C03641=1051.470,441.160,366.579,176.054,43.114,158.636
C03642=1051.459,440.916,366.630,176.041,43.103,158.631
C03643=1051.447,440.672,366.681,176.027,43.091,158.627
C03644=1051.435,440.427,366.732,176.014,43.081,158.623
C03645=1051.424,440.183,366.784,176.001,43.069,158.619
C03646=1051.413,439.938,366.835,175.987,43.058,158.615
C03647=1051.402,439.694,366.886,175.974,43.047,158.611
C03648=1051.390,439.450,366.937,175.961,43.036,158.607
C03649=1051.379,439.205,366.988,175.949,43.025,158.603
C03650=1051.364,438.882,367.055,175.931,43.011,158.597
C03651=1051.349,438.559,367.122,175.914,42.996,158.592
C03652=1051.334,438.236,367.189,175.897,42.981,158.587
C03653=1051.320,437.914,367.256,175.881,42.967,158.581
C03654=1051.308,437.669,367.307,175.868,42.956,158.577
C03655=1051.297,437.424,367.357,175.854,42.945,158.573
C03656=1051.286,437.180,367.408,175.843,42.935,158.570
C03657=1051.274,436.935,367.459,175.830,42.924,158.566
C03658=1051.263,436.691,367.509,175.818,42.913,158.562
C03659=1051.253,436.446,367.559,175.805,42.902,158.558
C03660=1051.242,436.201,367.609,175.792,42.892,158.554
C03661=1051.230,435.956,367.660,175.780,42.881,158.550
C03662=1051.219,435.712,367.710,175.767,42.871,158.546
C03663=1051.209,435.467,367.760,175.755,42.860,158.542
C03664=1051.198,435.222,367.810,175.742,42.850,158.539
C03665=1051.186,434.978,367.860,175.731,42.839,158.535
C03666=1051.175,434.733,367.910,175.719,42.829,158.531
C03667=1051.164,434.489,367.960,175.706,42.819,158.527
C03668=1051.154,434.244,368.009,175.694,42.808,158.524
C03669=1051.143,433.999,368.060,175.683,42.798,158.520
C03670=1051.132,433.754,368.109,175.670,42.788,158.516
C03671=1051.121,433.509,368.159,175.658,42.778,158.513
C03672=1051.110,433.264,368.208,175.647,42.767,158.509
C03673=1051.099,433.020,368.258,175.635,42.757,158.505
C03674=1051.085,432.691,368.324,175.619,42.743,158.500
C03675=1051.071,432.362,368.391,175.603,42.730,158.495
C03676=1051.057,432.033,368.458,175.588,42.716,158.491
C03677=1051.042,431.704,368.524,175.572,42.702,158.486
C03678=1051.031,431.459,368.573,175.560,42.693,158.482
C03679=1051.020,431.214,368.623,175.549,42.683,158.479
C03680=1051.011,430.969,368.672,175.537,42.672,158.475
C03681=1051.000,430.724,368.721,175.526,42.663,158.472
C03682=1050.989,430.479,368.770,175.514,42.653,158.468
C03683=1050.978,430.235,368.819,175.503,42.643,158.465
C03684=1050.968,429.989,368.868,175.492,42.633,158.461
C03685=1050.958,429.745,368.918,175.480,42.623,158.458
C03686=1050.948,429.499,368.966,175.469,42.613,158.454
C03687=1050.937,429.255,369.015,175.458,42.604,158.451
C03688=1050.927,429.010,369.064,175.447,42.594,158.447
C03689=1050.915,428.764,369.112,175.436,42.584,158.444
C03690=1050.906,428.519,369.161,175.425,42.575,158.440
C03691=1050.894,428.275,369.210,175.414,42.565,158.437
C03692=1050.885,428.030,369.258,175.403,42.555,158.434
C03693=1050.874,427.784,369.307,175.392,42.546,158.430
C03694=1050.864,427.539,369.355,175.380,42.536,158.427
C03695=1050.854,427.294,369.404,175.370,42.526,158.424
C03696=1050.843,427.049,369.452,175.359,42.517,158.420
C03697=1050.833,426.804,369.501,175.348,42.507,158.417
C03698=1050.823,426.559,369.548,175.338,42.498,158.414
C03699=1050.812,426.314,369.597,175.327,42.489,158.411
C03700=1050.802,426.069,369.645,175.316,42.480,158.407
C03701=1050.792,425.823,369.693,175.306,42.470,158.404
C03702=1050.782,425.579,369.741,175.295,42.461,158.401
C03703=1050.772,425.334,369.790,175.285,42.451,158.397
C03704=1050.761,425.088,369.837,175.274,42.442,158.394
C03705=1050.751,424.843,369.886,175.263,42.433,158.391
C03706=1050.741,424.597,369.933,175.253,42.424,158.388
C03707=1050.731,424.353,369.981,175.242,42.415,158.385
C03708=1050.721,424.108,370.028,175.232,42.405,158.382
C03709=1050.710,423.861,370.076,175.221,42.397,158.378
C03710=1050.700,423.617,370.124,175.211,42.387,158.375
C03711=1050.690,423.371,370.171,175.200,42.378,158.372
C03712=1050.680,423.126,370.219,175.191,42.369,158.369
C03713=1050.670,422.880,370.266,175.181,42.360,158.366
C03714=1050.660,422.636,370.314,175.170,42.351,158.363
C03715=1050.649,422.390,370.362,175.160,42.342,158.360
C03716=1050.640,422.145,370.409,175.149,42.333,158.357
C03717=1050.630,421.900,370.457,175.140,42.324,158.354
C03718=1050.620,421.655,370.503,175.130,42.315,158.351
C03719=1050.610,421.410,370.551,175.119,42.307,158.348
C03720=1050.601,421.164,370.598,175.109,42.298,158.345
C03721=1050.590,420.919,370.646,175.100,42.289,158.342
C03722=1050.581,420.673,370.692,175.090,42.280,158.339
C03723=1050.570,420.428,370.739,175.079,42.271,158.335
C03724=1050.561,420.183,370.787,175.070,42.262,158.332
C03725=1050.551,419.937,370.834,175.060,42.253,158.329
C03726=1050.541,419.692,370.881,175.050,42.245,158.327
C03727=1050.531,419.446,370.928,175.041,42.236,158.324
C03728=1050.523,419.201,370.974,175.030,42.228,158.321
C03729=1050.512,418.955,371.022,175.021,42.219,158.318
C03730=1050.496,418.571,371.095,175.006,42.205,158.313
C03731=1050.481,418.186,371.168,174.991,42.192,158.309
C03732=1050.466,417.802,371.240,174.976,42.179,158.304
C03733=1050.451,417.417,371.313,174.961,42.166,158.300
C03734=1050.441,417.171,371.360,174.951,42.157,158.297
C03735=1050.432,416.926,371.406,174.942,42.149,158.294
C03736=1050.422,416.680,371.453,174.933,42.141,158.291
C03737=1050.413,416.434,371.499,174.923,42.132,158.288
C03738=1050.403,416.189,371.546,174.914,42.124,158.286
C03739=1050.393,415.944,371.592,174.904,42.115,158.283
C03740=1050.384,415.697,371.638,174.895,42.107,158.280
C03741=1050.374,415.452,371.684,174.886,42.099,158.277
C03742=1050.365,415.207,371.730,174.877,42.090,158.275
C03743=1050.355,414.961,371.777,174.868,42.082,158.272
C03744=1050.345,414.716,371.822,174.859,42.074,158.269
C03745=1050.335,414.470,371.869,174.849,42.066,158.266
C03746=1050.326,414.225,371.914,174.840,42.057,158.264
C03747=1050.317,413.979,371.960,174.831,42.050,158.261
C03748=1050.308,413.734,372.006,174.821,42.042,158.258
C03749=1050.298,413.488,372.052,174.813,42.033,158.256
C03750=1050.289,413.242,372.098,174.804,42.025,158.253
C03751=1050.280,412.997,372.144,174.795,42.017,158.250
C03752=1050.271,412.751,372.190,174.786,42.009,158.247
C03753=1050.260,412.505,372.235,174.777,42.001,158.245
C03754=1050.251,412.259,372.280,174.768,41.993,158.242
C03755=1050.242,412.014,372.326,174.759,41.986,158.240
C03756=1050.232,411.769,372.371,174.750,41.978,158.237
C03757=1050.223,411.522,372.417,174.742,41.970,158.234
C03758=1050.213,411.277,372.462,174.733,41.962,158.232
C03759=1050.204,411.031,372.508,174.724,41.954,158.229
C03760=1050.195,410.786,372.553,174.715,41.946,158.227
C03761=1050.185,410.540,372.598,174.707,41.939,158.224
C03762=1050.176,410.294,372.644,174.697,41.931,158.222
C03763=1050.166,410.049,372.689,174.689,41.923,158.219
C03764=1050.157,409.803,372.734,174.680,41.915,158.216
C03765=1050.148,409.557,372.779,174.672,41.907,158.214
C03766=1050.139,409.312,372.824,174.663,41.899,158.211
C03767=1050.130,409.065,372.869,174.655,41.892,158.209
C03768=1050.120,408.820,372.914,174.646,41.884,158.206
C03769=1050.111,408.574,372.959,174.638,41.877,158.204
C03770=1050.102,408.328,373.004,174.629,41.869,158.201
C03771=1050.093,408.082,373.049,174.621,41.861,158.199
C03772=1050.083,407.836,373.094,174.612,41.854,158.196
C03773=1050.075,407.591,373.139,174.604,41.846,158.194
C03774=1050.066,407.345,373.184,174.595,41.839,158.191
C03775=1050.056,407.099,373.228,174.588,41.831,158.189
C03776=1050.048,406.853,373.274,174.579,41.824,158.187
C03777=1050.038,406.607,373.318,174.571,41.817,158.184
C03778=1050.030,406.362,373.363,174.562,41.809,158.182
C03779=1050.020,406.116,373.407,174.554,41.801,158.179
C03780=1050.011,405.870,373.452,174.546,41.794,158.177
C03781=1050.003,405.625,373.496,174.537,41.787,158.175
C03782=1049.994,405.378,373.541,174.529,41.779,158.172
C03783=1049.984,405.133,373.585,174.522,41.772,158.170
C03784=1049.976,404.887,373.630,174.513,41.765,158.167
C03785=1049.967,404.641,373.674,174.505,41.757,158.165
C03786=1049.953,404.263,373.742,174.493,41.746,158.161
C03787=1049.939,403.885,373.811,174.480,41.735,158.158
C03788=1049.925,403.507,373.878,174.468,41.724,158.154
C03789=1049.912,403.129,373.946,174.456,41.712,158.151
C03790=1049.903,402.883,373.990,174.447,41.705,158.148
C03791=1049.894,402.637,374.034,174.440,41.698,158.146
C03792=1049.886,402.391,374.079,174.432,41.691,158.144
C03793=1049.876,402.145,374.123,174.424,41.684,158.141
C03794=1049.868,401.899,374.166,174.417,41.677,158.139
C03795=1049.858,401.653,374.210,174.408,41.670,158.137
C03796=1049.850,401.407,374.254,174.400,41.663,158.135
C03797=1049.841,401.161,374.298,174.393,41.656,158.132
C03798=1049.832,400.915,374.341,174.385,41.649,158.130
C03799=1049.823,400.670,374.385,174.377,41.642,158.128
C03800=1049.814,400.423,374.428,174.370,41.635,158.126
C03801=1049.806,400.178,374.472,174.361,41.628,158.123
C03802=1049.796,399.931,374.516,174.354,41.621,158.121
C03803=1049.788,399.685,374.559,174.346,41.614,158.119
C03804=1049.779,399.440,374.603,174.338,41.608,158.117
C03805=1049.770,399.194,374.646,174.331,41.600,158.115
C03806=1049.762,398.947,374.690,174.323,41.594,158.113
C03807=1049.753,398.701,374.734,174.316,41.587,158.110
C03808=1049.745,398.455,374.777,174.308,41.580,158.108
C03809=1049.736,398.209,374.820,174.301,41.573,158.106
C03810=1049.727,397.963,374.864,174.293,41.566,158.104
C03811=1049.718,397.717,374.907,174.286,41.560,158.102
C03812=1049.710,397.471,374.950,174.278,41.553,158.100
C03813=1049.701,397.225,374.993,174.271,41.546,158.097
C03814=1049.692,396.980,375.037,174.263,41.539,158.095
C03815=1049.684,396.734,375.080,174.256,41.533,158.093
C03816=1049.675,396.487,375.123,174.248,41.526,158.091
C03817=1049.667,396.241,375.166,174.241,41.519,158.089
C03818=1049.658,395.995,375.209,174.233,41.513,158.087
C03819=1049.650,395.749,375.252,174.226,41.506,158.085
C03820=1049.641,395.504,375.294,174.219,41.499,158.083
C03821=1049.632,395.258,375.337,174.211,41.493,158.081
C03822=1049.623,395.011,375.381,174.204,41.486,158.078
C03823=1049.615,394.764,375.423,174.196,41.480,158.077
C03824=1049.607,394.519,375.466,174.189,41.473,158.074
C03825=1049.598,394.273,375.508,174.182,41.467,158.072
C03826=1049.589,394.027,375.551,174.175,41.460,158.070
C03827=1049.581,393.781,375.594,174.168,41.454,158.068
C03828=1049.573,393.534,375.637,174.161,41.447,158.066
C03829=1049.564,393.288,375.680,174.153,41.441,158.064
C03830=1049.556,393.042,375.723,174.146,41.435,158.062
C03831=1049.547,392.796,375.764,174.138,41.428,158.060
C03832=1049.538,392.550,375.807,174.131,41.422,158.058
C03833=1049.530,392.304,375.849,174.125,41.415,158.056
C03834=1049.522,392.058,375.892,174.118,41.409,158.054
C03835=1049.513,391.811,375.934,174.110,41.403,158.052
C03836=1049.505,391.565,375.977,174.103,41.396,158.050
C03837=1049.496,391.319,376.019,174.097,41.390,158.048
C03838=1049.487,391.073,376.062,174.090,41.384,158.046
C03839=1049.480,390.827,376.104,174.082,41.377,158.044
C03840=1049.471,390.580,376.146,174.075,41.371,158.042
C03841=1049.462,390.334,376.188,174.068,41.365,158.040
C03842=1049.450,389.975,376.250,174.058,41.356,158.038
C03843=1049.438,389.616,376.311,174.048,41.347,158.035
C03844=1049.426,389.256,376.372,174.038,41.338,158.032
C03845=1049.414,388.897,376.434,174.028,41.329,158.029
C03846=1049.406,388.650,376.476,174.021,41.323,158.027
C03847=1049.397,388.404,376.518,174.014,41.316,158.025
C03848=1049.389,388.157,376.560,174.007,41.310,158.023
C03849=1049.380,387.911,376.601,174.000,41.304,158.022
C03850=1049.371,387.665,376.643,173.994,41.299,158.020
C03851=1049.364,387.419,376.685,173.987,41.292,158.018
C03852=1049.355,387.172,376.726,173.980,41.286,158.016
C03853=1049.346,386.926,376.768,173.974,41.281,158.014
C03854=1049.339,386.680,376.810,173.967,41.274,158.012
C03855=1049.330,386.433,376.851,173.960,41.269,158.011
C03856=1049.322,386.187,376.893,173.953,41.263,158.009
C03857=1049.313,385.940,376.934,173.946,41.256,158.007
C03858=1049.305,385.695,376.976,173.940,41.251,158.005
C03859=1049.297,385.448,377.018,173.933,41.244,158.003
C03860=1049.289,385.202,377.058,173.927,41.239,158.001
C03861=1049.280,384.955,377.100,173.920,41.233,158.000
C03862=1049.273,384.709,377.141,173.913,41.227,157.998
C03863=1049.264,384.462,377.183,173.907,41.221,157.996
C03864=1049.256,384.216,377.224,173.900,41.216,157.994
C03865=1049.248,383.970,377.266,173.894,41.209,157.992
C03866=1049.239,383.723,377.307,173.887,41.204,157.991
C03867=1049.231,383.478,377.348,173.881,41.198,157.989
C03868=1049.224,383.231,377.389,173.874,41.192,157.987
C03869=1049.215,382.985,377.431,173.868,41.186,157.985
C03870=1049.207,382.738,377.472,173.861,41.181,157.983
C03871=1049.200,382.492,377.513,173.855,41.175,157.982
C03872=1049.191,382.245,377.554,173.848,41.169,157.980
C03873=1049.183,381.999,377.595,173.842,41.163,157.978
C03874=1049.175,381.752,377.636,173.836,41.158,157.976
C03875=1049.167,381.505,377.677,173.829,41.152,157.975
C03876=1049.159,381.259,377.718,173.823,41.146,157.973
C03877=1049.150,381.014,377.759,173.816,41.141,157.971
C03878=1049.143,380.767,377.801,173.810,41.135,157.969
C03879=1049.135,380.521,377.841,173.803,41.129,157.968
C03880=1049.126,380.274,377.882,173.797,41.124,157.966
C03881=1049.119,380.027,377.924,173.791,41.118,157.964
C03882=1049.111,379.781,377.964,173.784,41.112,157.963
C03883=1049.103,379.535,378.005,173.778,41.106,157.961
C03884=1049.095,379.288,378.045,173.772,41.101,157.959
C03885=1049.087,379.042,378.086,173.765,41.096,157.957
C03886=1049.079,378.794,378.126,173.760,41.090,157.956
C03887=1049.071,378.548,378.167,173.753,41.085,157.954
C03888=1049.063,378.302,378.208,173.747,41.079,157.952
C03889=1049.055,378.055,378.248,173.741,41.074,157.951
C03890=1049.047,377.809,378.288,173.734,41.068,157.949
C03891=1049.039,377.562,378.329,173.728,41.063,157.948
C03892=1049.031,377.316,378.369,173.722,41.057,157.946
C03893=1049.022,377.068,378.410,173.715,41.052,157.944
C03894=1049.014,376.822,378.450,173.710,41.046,157.942
C03895=1049.006,376.576,378.491,173.704,41.041,157.941
C03896=1048.999,376.329,378.531,173.698,41.036,157.939
C03897=1048.991,376.083,378.572,173.691,41.030,157.938
C03898=1048.980,375.756,378.624,173.684,41.023,157.936
C03899=1048.970,375.430,378.678,173.675,41.016,157.933
C03900=1048.959,375.103,378.731,173.667,41.009,157.931
C03901=1048.949,374.776,378.784,173.660,41.002,157.929
C03902=1048.941,374.530,378.825,173.654,40.997,157.928
C03903=1048.933,374.283,378.865,173.647,40.992,157.926
C03904=1048.925,374.036,378.905,173.641,40.986,157.924
C03905=1048.917,373.790,378.945,173.635,40.981,157.923
C03906=1048.910,373.543,378.985,173.630,40.975,157.921
C03907=1048.902,373.297,379.025,173.624,40.970,157.920
C03908=1048.894,373.050,379.064,173.617,40.965,157.918
C03909=1048.886,372.804,379.105,173.611,40.960,157.916
C03910=1048.878,372.557,379.145,173.606,40.955,157.915
C03911=1048.871,372.310,379.184,173.600,40.949,157.913
C03912=1048.863,372.064,379.224,173.594,40.944,157.912
C03913=1048.856,371.817,379.264,173.588,40.939,157.910
C03914=1048.848,371.570,379.304,173.582,40.934,157.909
C03915=1048.840,371.323,379.344,173.576,40.928,157.907
C03916=1048.832,371.076,379.383,173.570,40.923,157.905
C03917=1048.825,370.830,379.423,173.565,40.918,157.904
C03918=1048.817,370.583,379.463,173.559,40.913,157.902
C03919=1048.809,370.337,379.502,173.553,40.908,157.901
C03920=1048.801,370.090,379.542,173.548,40.903,157.900
C03921=1048.792,369.843,379.581,173.542,40.898,157.898
C03922=1048.786,369.596,379.620,173.535,40.893,157.896
C03923=1048.778,369.349,379.660,173.530,40.888,157.895
C03924=1048.769,369.103,379.699,173.524,40.883,157.893
C03925=1048.762,368.857,379.739,173.518,40.878,157.892
C03926=1048.754,368.609,379.777,173.513,40.873,157.890
C03927=1048.746,368.362,379.817,173.507,40.868,157.889
C03928=1048.738,368.116,379.857,173.501,40.863,157.887
C03929=1048.731,367.869,379.895,173.496,40.858,157.886
C03930=1048.723,367.622,379.935,173.490,40.853,157.885
C03931=1048.716,367.376,379.974,173.485,40.848,157.883
C03932=1048.708,367.129,380.013,173.479,40.843,157.882
C03933=1048.700,366.882,380.053,173.473,40.838,157.880
C03934=1048.693,366.635,380.092,173.468,40.834,157.879
C03935=1048.684,366.389,380.131,173.462,40.828,157.877
C03936=1048.678,366.142,380.170,173.456,40.824,157.876
C03937=1048.669,365.895,380.209,173.451,40.818,157.874
C03938=1048.662,365.648,380.248,173.445,40.814,157.873
C03939=1048.655,365.401,380.287,173.440,40.809,157.871
C03940=1048.646,365.154,380.327,173.434,40.804,157.870
C03941=1048.640,364.908,380.365,173.428,40.799,157.869
C03942=1048.631,364.661,380.405,173.423,40.794,157.867
C03943=1048.624,364.414,380.444,173.417,40.790,157.866
C03944=1048.617,364.168,380.482,173.412,40.785,157.864
C03945=1048.609,363.920,380.521,173.406,40.780,157.863
C03946=1048.602,363.674,380.560,173.401,40.775,157.862
C03947=1048.594,363.427,380.599,173.395,40.770,157.860
C03948=1048.587,363.180,380.637,173.390,40.765,157.859
C03949=1048.579,362.933,380.677,173.385,40.761,157.857
C03950=1048.572,362.686,380.715,173.379,40.756,157.856
C03951=1048.564,362.440,380.753,173.374,40.751,157.854
C03952=1048.557,362.192,380.792,173.368,40.746,157.853
C03953=1048.549,361.946,380.830,173.363,40.742,157.852
C03954=1048.540,361.638,380.879,173.356,40.736,157.850
C03955=1048.529,361.330,380.927,173.349,40.730,157.848
C03956=1048.520,361.023,380.975,173.342,40.724,157.846
C03957=1048.511,360.715,381.023,173.336,40.719,157.845
C03958=1048.504,360.468,381.061,173.331,40.714,157.844
C03959=1048.496,360.222,381.099,173.326,40.710,157.842
C03960=1048.488,359.975,381.138,173.320,40.705,157.841
C03961=1048.480,359.728,381.176,173.315,40.700,157.839
C03962=1048.474,359.481,381.214,173.309,40.696,157.838
C03963=1048.466,359.234,381.253,173.304,40.691,157.837
C03964=1048.458,358.987,381.291,173.299,40.686,157.835
C03965=1048.451,358.741,381.329,173.294,40.682,157.834
C03966=1048.443,358.493,381.367,173.288,40.678,157.833
C03967=1048.436,358.246,381.406,173.283,40.673,157.831
C03968=1048.429,357.999,381.444,173.277,40.669,157.830
C03969=1048.421,357.752,381.482,173.273,40.664,157.829
C03970=1048.414,357.506,381.520,173.268,40.660,157.827
C03971=1048.406,357.258,381.559,173.262,40.655,157.826
C03972=1048.398,357.011,381.596,173.257,40.651,157.825
C03973=1048.391,356.764,381.634,173.252,40.646,157.823
C03974=1048.384,356.518,381.672,173.247,40.642,157.822
C03975=1048.376,356.270,381.710,173.241,40.637,157.821
C03976=1048.368,356.023,381.748,173.236,40.633,157.820
C03977=1048.361,355.776,381.786,173.231,40.628,157.818
C03978=1048.353,355.530,381.824,173.226,40.624,157.817
C03979=1048.346,355.283,381.861,173.221,40.619,157.816
C03980=1048.339,355.035,381.899,173.215,40.615,157.814
C03981=1048.331,354.789,381.937,173.210,40.611,157.813
C03982=1048.323,354.541,381.975,173.206,40.606,157.812
C03983=1048.316,354.294,382.013,173.200,40.602,157.811
C03984=1048.309,354.047,382.050,173.195,40.597,157.809
C03985=1048.301,353.800,382.088,173.191,40.593,157.808
C03986=1048.294,353.553,382.126,173.185,40.589,157.807
C03987=1048.287,353.306,382.163,173.180,40.585,157.806
C03988=1048.280,353.059,382.201,173.175,40.580,157.804
C03989=1048.272,352.812,382.238,173.170,40.575,157.803
C03990=1048.265,352.565,382.277,173.165,40.571,157.802
C03991=1048.258,352.318,382.314,173.161,40.567,157.801
C03992=1048.250,352.071,382.352,173.155,40.563,157.799
C03993=1048.243,351.824,382.389,173.150,40.559,157.798
C03994=1048.236,351.577,382.427,173.146,40.554,157.797
C03995=1048.229,351.330,382.464,173.140,40.550,157.796
C03996=1048.221,351.082,382.502,173.135,40.545,157.794
C03997=1048.214,350.835,382.539,173.130,40.541,157.793
C03998=1048.207,350.588,382.577,173.125,40.537,157.792
C03999=1048.199,350.341,382.614,173.120,40.533,157.791
C04000=1048.192,350.094,382.651,173.115,40.528,157.789
C04001=1048.185,349.846,382.688,173.110,40.524,157.788
C04002=1048.178,349.599,382.726,173.106,40.520,157.787
C04003=1048.170,349.352,382.763,173.101,40.516,157.786
C04004=1048.163,349.106,382.800,173.095,40.512,157.785
C04005=1048.156,348.858,382.837,173.091,40.508,157.783
C04006=1048.149,348.611,382.874,173.086,40.503,157.782
C04007=1048.141,348.364,382.911,173.081,40.499,157.781
C04008=1048.134,348.117,382.949,173.076,40.495,157.780
C04009=1048.127,347.869,382.985,173.071,40.491,157.779
C04010=1048.117,347.568,383.031,173.065,40.486,157.777
C04011=1048.108,347.265,383.076,173.060,40.481,157.776
C04012=1048.100,346.963,383.121,173.053,40.476,157.774
C04013=1048.092,346.661,383.166,173.048,40.471,157.773
C04014=1048.084,346.415,383.203,173.043,40.467,157.772
C04015=1048.076,346.167,383.241,173.038,40.462,157.770
C04016=1048.069,345.920,383.277,173.033,40.459,157.769
C04017=1048.062,345.672,383.314,173.029,40.454,157.768
C04018=1048.055,345.426,383.351,173.023,40.450,157.767
C04019=1048.047,345.178,383.387,173.019,40.446,157.766
C04020=1048.040,344.931,383.424,173.014,40.442,157.765
C04021=1048.033,344.683,383.461,173.010,40.438,157.764
C04022=1048.026,344.437,383.498,173.005,40.434,157.762
C04023=1048.019,344.190,383.535,173.000,40.430,157.761
C04024=1048.011,343.942,383.571,172.995,40.426,157.760
C04025=1048.005,343.696,383.608,172.991,40.422,157.759
C04026=1047.997,343.448,383.644,172.986,40.418,157.758
C04027=1047.990,343.201,383.681,172.981,40.414,157.757
C04028=1047.984,342.953,383.718,172.976,40.410,157.755
C04029=1047.976,342.707,383.754,172.972,40.406,157.754
C04030=1047.969,342.459,383.791,172.968,40.402,157.753
C04031=1047.962,342.212,383.827,172.963,40.398,157.752
C04032=1047.955,341.964,383.864,172.958,40.394,157.751
C04033=1047.947,341.717,383.900,172.953,40.390,157.750
C04034=1047.940,341.470,383.936,172.949,40.387,157.749
C04035=1047.933,341.222,383.973,172.944,40.382,157.748
C04036=1047.925,340.975,384.009,172.940,40.379,157.747
C04037=1047.918,340.729,384.046,172.935,40.375,157.745
C04038=1047.911,340.481,384.082,172.930,40.371,157.744
C04039=1047.903,340.234,384.119,172.926,40.367,157.743
C04040=1047.897,339.986,384.154,172.921,40.363,157.742
C04041=1047.890,339.739,384.191,172.917,40.359,157.741
C04042=1047.883,339.492,384.226,172.912,40.355,157.740
C04043=1047.875,339.244,384.263,172.908,40.351,157.739
C04044=1047.869,338.997,384.299,172.903,40.348,157.738
C04045=1047.861,338.750,384.335,172.898,40.344,157.737
C04046=1047.854,338.503,384.371,172.894,40.340,157.736
C04047=1047.847,338.255,384.408,172.889,40.336,157.734
C04048=1047.840,338.009,384.444,172.885,40.332,157.733
C04049=1047.832,337.761,384.479,172.881,40.328,157.732
C04050=1047.826,337.514,384.516,172.876,40.325,157.731
C04051=1047.818,337.266,384.552,172.872,40.321,157.730
C04052=1047.811,337.019,384.588,172.867,40.317,157.729
C04053=1047.804,336.771,384.623,172.862,40.314,157.728
C04054=1047.798,336.524,384.660,172.858,40.310,157.727
C04055=1047.790,336.277,384.696,172.854,40.306,157.726
C04056=1047.783,336.030,384.732,172.849,40.302,157.725
C04057=1047.777,335.782,384.768,172.845,40.298,157.724
C04058=1047.769,335.535,384.804,172.841,40.295,157.723
C04059=1047.762,335.288,384.839,172.836,40.291,157.722
C04060=1047.755,335.040,384.875,172.831,40.287,157.721
C04061=1047.748,334.793,384.910,172.827,40.283,157.720
C04062=1047.740,334.545,384.946,172.822,40.280,157.718
C04063=1047.734,334.298,384.982,172.818,40.276,157.717
C04064=1047.726,334.051,385.017,172.814,40.272,157.716
C04065=1047.719,333.803,385.053,172.809,40.268,157.715
C04066=1047.710,333.497,385.097,172.804,40.264,157.714
C04067=1047.702,333.192,385.142,172.798,40.259,157.713
C04068=1047.693,332.886,385.185,172.793,40.255,157.712
C04069=1047.684,332.580,385.229,172.788,40.250,157.710
C04070=1047.677,332.333,385.264,172.784,40.247,157.709
C04071=1047.670,332.085,385.300,172.780,40.243,157.708
C04072=1047.663,331.838,385.335,172.774,40.240,157.707
C04073=1047.657,331.590,385.371,172.770,40.236,157.706
C04074=1047.649,331.343,385.407,172.766,40.232,157.705
C04075=1047.643,331.095,385.442,172.762,40.229,157.704
C04076=1047.636,330.848,385.477,172.758,40.225,157.703
C04077=1047.629,330.601,385.513,172.753,40.221,157.702
C04078=1047.622,330.352,385.548,172.749,40.217,157.701
C04079=1047.615,330.106,385.584,172.745,40.214,157.700
C04080=1047.608,329.858,385.619,172.741,40.210,157.699
C04081=1047.601,329.611,385.654,172.736,40.207,157.698
C04082=1047.593,329.364,385.689,172.732,40.203,157.697
C04083=1047.586,329.116,385.724,172.728,40.200,157.696
C04084=1047.579,328.868,385.759,172.724,40.196,157.695
C04085=1047.572,328.621,385.794,172.720,40.193,157.694
C04086=1047.564,328.373,385.829,172.715,40.189,157.693
C04087=1047.558,328.126,385.865,172.711,40.186,157.692
C04088=1047.550,327.879,385.899,172.707,40.182,157.691
C04089=1047.543,327.632,385.934,172.703,40.179,157.690
C04090=1047.537,327.384,385.969,172.698,40.176,157.689
C04091=1047.529,327.136,386.004,172.694,40.172,157.688
C04092=1047.522,326.888,386.039,172.690,40.168,157.687
C04093=1047.515,326.641,386.074,172.686,40.165,157.686
C04094=1047.508,326.394,386.108,172.682,40.161,157.685
C04095=1047.501,326.147,386.144,172.678,40.158,157.684
C04096=1047.494,325.900,386.178,172.673,40.155,157.683
C04097=1047.486,325.651,386.213,172.669,40.151,157.683
C04098=1047.480,325.404,386.248,172.665,40.148,157.682
C04099=1047.472,325.157,386.283,172.661,40.144,157.681
C04100=1047.465,324.909,386.318,172.657,40.141,157.680
C04101=1047.458,324.661,386.352,172.653,40.138,157.679
C04102=1047.451,324.414,386.387,172.648,40.134,157.678
C04103=1047.445,324.167,386.422,172.644,40.131,157.677
C04104=1047.437,323.919,386.456,172.640,40.128,157.676
C04105=1047.431,323.672,386.491,172.636,40.124,157.675
C04106=1047.423,323.425,386.525,172.632,40.121,157.674
C04107=1047.417,323.177,386.560,172.628,40.117,157.673
C04108=1047.409,322.930,386.594,172.624,40.113,157.672
C04109=1047.403,322.682,386.629,172.620,40.110,157.671
C04110=1047.396,322.434,386.664,172.616,40.107,157.670
C04111=1047.389,322.187,386.698,172.611,40.104,157.669
C04112=1047.382,321.939,386.733,172.607,40.100,157.668
C04113=1047.375,321.692,386.767,172.603,40.097,157.667
C04114=1047.368,321.444,386.802,172.599,40.094,157.666
C04115=1047.361,321.197,386.836,172.595,40.090,157.666
C04116=1047.354,320.949,386.871,172.591,40.086,157.665
C04117=1047.348,320.701,386.905,172.587,40.083,157.664
C04118=1047.340,320.454,386.940,172.583,40.080,157.663
C04119=1047.334,320.206,386.974,172.579,40.077,157.662
C04120=1047.326,319.959,387.009,172.575,40.073,157.661
C04121=1047.320,319.711,387.043,172.571,40.070,157.660
C04122=1047.311,319.400,387.085,172.566,40.066,157.659
C04123=1047.303,319.090,387.129,172.561,40.062,157.658
C04124=1047.294,318.779,387.172,172.556,40.057,157.656
C04125=1047.285,318.468,387.216,172.552,40.053,157.655
C04126=1047.278,318.220,387.250,172.548,40.050,157.654
C04127=1047.272,317.973,387.284,172.544,40.046,157.654
C04128=1047.265,317.725,387.318,172.540,40.043,157.653
C04129=1047.258,317.478,387.353,172.536,40.040,157.652
C04130=1047.251,317.230,387.387,172.532,40.037,157.651
C04131=1047.245,316.983,387.421,172.528,40.033,157.650
C04132=1047.238,316.735,387.454,172.524,40.030,157.649
C04133=1047.232,316.487,387.489,172.520,40.027,157.648
C04134=1047.225,316.252,387.522,172.516,40.024,157.647
C04135=1047.219,316.017,387.554,172.513,40.020,157.646
C04136=1047.212,315.782,387.586,172.509,40.017,157.645
C04137=1047.206,315.546,387.618,172.505,40.014,157.645
C04138=1047.199,315.311,387.651,172.502,40.011,157.644
C04139=1047.193,315.075,387.683,172.498,40.008,157.643
C04140=1047.187,314.840,387.716,172.494,40.004,157.642
C04141=1047.181,314.605,387.748,172.490,40.002,157.641
C04142=1047.174,314.357,387.782,172.486,39.999,157.640
C04143=1047.167,314.110,387.815,172.483,39.995,157.640
C04144=1047.161,313.862,387.850,172.479,39.992,157.639
C04145=1047.153,313.615,387.884,172.476,39.989,157.638
C04146=1047.148,313.367,387.918,172.472,39.985,157.637
C04147=1047.140,313.120,387.951,172.468,39.982,157.636
C04148=1047.135,312.872,387.985,172.464,39.979,157.635
C04149=1047.127,312.625,388.019,172.460,39.976,157.634
C04150=1047.120,312.377,388.053,172.456,39.972,157.633
C04151=1047.113,312.129,388.087,172.452,39.969,157.632
C04152=1047.107,311.882,388.120,172.448,39.966,157.632
C04153=1047.099,311.634,388.154,172.445,39.963,157.631
C04154=1047.092,311.386,388.187,172.441,39.960,157.630
C04155=1047.086,311.139,388.221,172.437,39.957,157.629
C04156=1047.079,310.891,388.254,172.433,39.954,157.628
C04157=1047.071,310.644,388.287,172.429,39.951,157.627
C04158=1047.064,310.397,388.321,172.425,39.947,157.626
C04159=1047.057,310.149,388.354,172.422,39.945,157.626
C04160=1047.050,309.901,388.388,172.419,39.941,157.625
C04161=1047.044,309.653,388.420,172.415,39.938,157.624
C04162=1047.037,309.406,388.454,172.411,39.935,157.623
C04163=1047.029,309.158,388.488,172.407,39.932,157.622
C04164=1047.023,308.910,388.521,172.403,39.929,157.621
C04165=1047.016,308.663,388.554,172.399,39.926,157.621
C04166=1047.010,308.415,388.587,172.395,39.923,157.620
C04167=1047.002,308.168,388.620,172.392,39.920,157.619
C04168=1046.995,307.920,388.653,172.388,39.917,157.618
C04169=1046.988,307.672,388.687,172.385,39.914,157.617
C04170=1046.981,307.424,388.720,172.381,39.911,157.617
C04171=1046.975,307.177,388.754,172.377,39.908,157.616
C04172=1046.968,306.929,388.787,172.373,39.904,157.615
C04173=1046.961,306.682,388.820,172.370,39.902,157.614
C04174=1046.954,306.434,388.853,172.366,39.898,157.613
C04175=1046.948,306.186,388.886,172.362,39.896,157.612
C04176=1046.940,305.939,388.919,172.359,39.892,157.612
C04177=1046.934,305.691,388.952,172.355,39.890,157.611
C04178=1046.925,305.360,388.996,172.350,39.885,157.610
C04179=1046.916,305.028,389.041,172.345,39.881,157.609
C04180=1046.907,304.698,389.085,172.340,39.877,157.607
C04181=1046.898,304.367,389.129,172.336,39.873,157.606
C04182=1046.892,304.119,389.162,172.332,39.870,157.605
C04183=1046.884,303.871,389.195,172.328,39.867,157.605
C04184=1046.878,303.624,389.227,172.324,39.864,157.604
C04185=1046.870,303.376,389.261,172.322,39.861,157.603
C04186=1046.864,303.128,389.294,172.318,39.858,157.602
C04187=1046.858,302.881,389.327,172.314,39.855,157.602
C04188=1046.851,302.633,389.360,172.310,39.852,157.601
C04189=1046.844,302.385,389.392,172.306,39.849,157.600
C04190=1046.837,302.138,389.426,172.303,39.846,157.599
C04191=1046.830,301.890,389.458,172.300,39.843,157.598
C04192=1046.824,301.642,389.491,172.296,39.840,157.597
C04193=1046.817,301.394,389.524,172.292,39.837,157.597
C04194=1046.811,301.147,389.557,172.289,39.834,157.596
C04195=1046.804,300.899,389.589,172.285,39.831,157.595
C04196=1046.798,300.652,389.622,172.282,39.828,157.594
C04197=1046.791,300.403,389.655,172.278,39.825,157.593
C04198=1046.784,300.156,389.688,172.275,39.822,157.593
C04199=1046.778,299.908,389.720,172.271,39.819,157.592
C04200=1046.771,299.660,389.753,172.267,39.816,157.591
C04201=1046.764,299.413,389.786,172.265,39.813,157.590
C04202=1046.758,299.165,389.818,172.261,39.809,157.589
C04203=1046.752,298.917,389.851,172.257,39.807,157.589
C04204=1046.745,298.669,389.884,172.254,39.804,157.588
C04205=1046.738,298.422,389.916,172.250,39.801,157.587
C04206=1046.731,298.174,389.949,172.247,39.798,157.586
C04207=1046.725,297.927,389.982,172.243,39.795,157.585
C04208=1046.719,297.679,390.015,172.240,39.792,157.585
C04209=1046.712,297.430,390.047,172.236,39.789,157.584
C04210=1046.705,297.183,390.079,172.232,39.786,157.583
C04211=1046.699,296.935,390.112,172.230,39.783,157.582
C04212=1046.693,296.688,390.145,172.226,39.780,157.581
C04213=1046.686,296.440,390.177,172.222,39.777,157.581
C04214=1046.680,296.193,390.210,172.219,39.774,157.580
C04215=1046.673,295.944,390.242,172.215,39.771,157.579
C04216=1046.666,295.696,390.275,172.212,39.768,157.578
C04217=1046.659,295.449,390.307,172.209,39.765,157.578
C04218=1046.653,295.201,390.339,172.205,39.762,157.577
C04219=1046.646,294.954,390.371,172.201,39.759,157.576
C04220=1046.639,294.705,390.404,172.199,39.757,157.575
C04221=1046.633,294.457,390.436,172.195,39.754,157.575
C04222=1046.626,294.210,390.468,172.192,39.750,157.574
C04223=1046.620,293.962,390.500,172.188,39.748,157.573
C04224=1046.613,293.714,390.533,172.185,39.745,157.572
C04225=1046.606,293.467,390.565,172.182,39.742,157.571
C04226=1046.599,293.218,390.596,172.178,39.740,157.571
C04227=1046.593,292.971,390.629,172.174,39.736,157.570
C04228=1046.586,292.723,390.661,172.171,39.733,157.569
C04229=1046.579,292.476,390.693,172.168,39.731,157.568
C04230=1046.573,292.227,390.725,172.164,39.728,157.568
C04231=1046.566,291.979,390.756,172.161,39.725,157.567
C04232=1046.559,291.732,390.788,172.158,39.722,157.566
C04233=1046.553,291.483,390.821,172.155,39.719,157.565
C04234=1046.545,291.194,390.858,172.150,39.716,157.564
C04235=1046.538,290.903,390.895,172.146,39.713,157.564
C04236=1046.530,290.613,390.932,172.142,39.709,157.563
C04237=1046.521,290.324,390.970,172.138,39.706,157.562
C04238=1046.515,290.076,391.002,172.135,39.703,157.561
C04239=1046.509,289.828,391.034,172.132,39.700,157.560
C04240=1046.502,289.580,391.065,172.129,39.698,157.560
C04241=1046.495,289.332,391.097,172.125,39.695,157.559
C04242=1046.489,289.084,391.129,172.122,39.692,157.558
C04243=1046.482,288.835,391.161,172.119,39.689,157.557
C04244=1046.475,288.588,391.193,172.115,39.687,157.557
C04245=1046.468,288.340,391.225,172.112,39.684,157.556
C04246=1046.462,288.092,391.257,172.109,39.681,157.555
C04247=1046.455,287.844,391.288,172.106,39.678,157.555
C04248=1046.448,287.596,391.320,172.102,39.675,157.554
C04249=1046.442,287.348,391.351,172.098,39.672,157.553
C04250=1046.435,287.101,391.383,172.096,39.669,157.552
C04251=1046.428,286.853,391.415,172.092,39.667,157.552
C04252=1046.421,286.605,391.446,172.089,39.664,157.551
C04253=1046.415,286.357,391.478,172.086,39.662,157.550
C04254=1046.408,286.110,391.509,172.083,39.659,157.549
C04255=1046.402,285.861,391.541,172.079,39.656,157.549
C04256=1046.395,285.613,391.573,172.076,39.653,157.548
C04257=1046.388,285.365,391.604,172.073,39.651,157.547
C04258=1046.382,285.118,391.635,172.070,39.648,157.547
C04259=1046.375,284.870,391.667,172.066,39.645,157.546
C04260=1046.368,284.622,391.698,172.064,39.642,157.545
C04261=1046.361,284.374,391.730,172.060,39.639,157.544
C04262=1046.355,284.126,391.761,172.056,39.637,157.544
C04263=1046.349,283.879,391.792,172.053,39.634,157.543
C04264=1046.342,283.631,391.824,172.050,39.631,157.542
C04265=1046.335,283.382,391.854,172.047,39.628,157.542
C04266=1046.329,283.134,391.886,172.043,39.626,157.541
C04267=1046.322,282.887,391.917,172.041,39.623,157.540
C04268=1046.315,282.639,391.949,172.038,39.620,157.539
C04269=1046.309,282.391,391.980,172.034,39.617,157.539
C04270=1046.302,282.143,392.012,172.031,39.614,157.538
C04271=1046.295,281.895,392.043,172.028,39.612,157.537
C04272=1046.289,281.646,392.074,172.025,39.609,157.537
C04273=1046.283,281.399,392.105,172.021,39.607,157.536
C04274=1046.276,281.151,392.136,172.019,39.604,157.535
C04275=1046.269,280.903,392.168,172.015,39.601,157.534
C04276=1046.263,280.655,392.198,172.012,39.598,157.534
C04277=1046.256,280.407,392.230,172.009,39.596,157.533
C04278=1046.249,280.159,392.261,172.006,39.593,157.532
C04279=1046.243,279.912,392.292,172.002,39.590,157.532
C04280=1046.237,279.663,392.323,172.000,39.587,157.531
C04281=1046.230,279.415,392.354,171.997,39.584,157.530
C04282=1046.223,279.168,392.386,171.993,39.582,157.529
C04283=1046.217,278.919,392.417,171.991,39.579,157.529
C04284=1046.210,278.671,392.448,171.987,39.577,157.528
C04285=1046.204,278.424,392.478,171.984,39.574,157.527
C04286=1046.197,278.176,392.509,171.980,39.571,157.527
C04287=1046.190,277.928,392.541,171.978,39.568,157.526
C04288=1046.184,277.679,392.571,171.975,39.566,157.525
C04289=1046.177,277.431,392.603,171.971,39.563,157.525
C04290=1046.170,277.153,392.637,171.968,39.560,157.524
C04291=1046.163,276.875,392.671,171.965,39.557,157.523
C04292=1046.155,276.596,392.707,171.961,39.554,157.522
C04293=1046.147,276.318,392.741,171.957,39.551,157.521
C04294=1046.141,276.069,392.772,171.955,39.548,157.521
C04295=1046.134,275.822,392.802,171.951,39.546,157.520
C04296=1046.127,275.573,392.833,171.948,39.543,157.519
C04297=1046.121,275.326,392.864,171.946,39.540,157.519
C04298=1046.115,275.077,392.895,171.942,39.537,157.518
C04299=1046.107,274.829,392.925,171.939,39.535,157.517
C04300=1046.101,274.582,392.956,171.937,39.532,157.517
C04301=1046.095,274.333,392.987,171.933,39.530,157.516
C04302=1046.088,274.085,393.017,171.930,39.527,157.515
C04303=1046.081,273.837,393.048,171.927,39.524,157.515
C04304=1046.075,273.589,393.079,171.924,39.522,157.514
C04305=1046.068,273.341,393.109,171.921,39.519,157.513
C04306=1046.061,273.093,393.140,171.918,39.516,157.513
C04307=1046.056,272.845,393.171,171.915,39.514,157.512
C04308=1046.048,272.597,393.201,171.912,39.511,157.511
C04309=1046.042,272.349,393.231,171.909,39.508,157.511
C04310=1046.036,272.102,393.263,171.906,39.506,157.510
C04311=1046.029,271.853,393.293,171.903,39.503,157.509
C04312=1046.022,271.605,393.323,171.900,39.501,157.509
C04313=1046.016,271.357,393.354,171.897,39.498,157.508
C04314=1046.009,271.109,393.384,171.894,39.495,157.507
C04315=1046.003,270.860,393.415,171.891,39.493,157.506
C04316=1045.996,270.613,393.445,171.888,39.490,157.506
C04317=1045.990,270.365,393.476,171.885,39.487,157.505
C04318=1045.982,270.117,393.506,171.882,39.485,157.504
C04319=1045.977,269.869,393.536,171.879,39.482,157.504
C04320=1045.969,269.621,393.566,171.876,39.479,157.503
C04321=1045.963,269.372,393.597,171.873,39.477,157.502
C04322=1045.956,269.125,393.627,171.870,39.474,157.502
C04323=1045.950,268.876,393.658,171.867,39.471,157.501
C04324=1045.944,268.628,393.687,171.864,39.469,157.500
C04325=1045.937,268.380,393.718,171.861,39.466,157.500
C04326=1045.930,268.132,393.748,171.858,39.463,157.499
C04327=1045.924,267.884,393.778,171.856,39.461,157.498
C04328=1045.917,267.636,393.809,171.852,39.458,157.498
C04329=1045.910,267.388,393.838,171.850,39.456,157.497
C04330=1045.904,267.140,393.869,171.847,39.453,157.496
C04331=1045.897,266.892,393.899,171.843,39.451,157.496
C04332=1045.890,266.644,393.929,171.841,39.448,157.495
C04333=1045.884,266.395,393.959,171.838,39.445,157.494
C04334=1045.878,266.147,393.989,171.835,39.443,157.494
C04335=1045.870,265.899,394.019,171.832,39.440,157.493
C04336=1045.865,265.651,394.049,171.829,39.438,157.492
C04337=1045.857,265.403,394.079,171.827,39.435,157.492
C04338=1045.852,265.155,394.110,171.824,39.432,157.491
C04339=1045.845,264.906,394.139,171.820,39.430,157.491
C04340=1045.838,264.659,394.169,171.818,39.427,157.490
C04341=1045.832,264.410,394.200,171.815,39.425,157.489
C04342=1045.825,264.163,394.229,171.812,39.422,157.489
C04343=1045.818,263.915,394.259,171.809,39.420,157.488
C04344=1045.813,263.666,394.289,171.806,39.417,157.487
C04345=1045.805,263.418,394.319,171.803,39.414,157.487
C04346=1045.799,263.144,394.352,171.800,39.412,157.486
C04347=1045.791,262.870,394.386,171.797,39.409,157.485
C04348=1045.784,262.596,394.419,171.793,39.406,157.484
C04349=1045.776,262.322,394.451,171.791,39.403,157.484
C04350=1045.769,262.073,394.481,171.788,39.400,157.483
C04351=1045.763,261.825,394.510,171.785,39.398,157.483
C04352=1045.756,261.577,394.540,171.782,39.395,157.482
C04353=1045.750,261.329,394.569,171.779,39.393,157.481
C04354=1045.743,261.081,394.599,171.777,39.390,157.481
C04355=1045.736,260.833,394.629,171.774,39.388,157.480
C04356=1045.729,260.584,394.658,171.770,39.386,157.479
C04357=1045.723,260.337,394.688,171.768,39.383,157.479
C04358=1045.716,260.088,394.717,171.765,39.381,157.478
C04359=1045.709,259.840,394.746,171.763,39.378,157.477
C04360=1045.702,259.592,394.777,171.760,39.376,157.477
C04361=1045.696,259.343,394.806,171.756,39.373,157.476
C04362=1045.689,259.095,394.836,171.754,39.371,157.476
C04363=1045.683,258.847,394.865,171.751,39.368,157.475
C04364=1045.675,258.599,394.895,171.749,39.365,157.474
C04365=1045.669,258.351,394.924,171.746,39.363,157.474
C04366=1045.663,258.103,394.953,171.742,39.360,157.473
C04367=1045.656,257.854,394.983,171.740,39.358,157.472
C04368=1045.650,257.606,395.012,171.737,39.355,157.472
C04369=1045.643,257.357,395.042,171.735,39.353,157.471
C04370=1045.636,257.110,395.071,171.732,39.350,157.470
C04371=1045.629,256.862,395.100,171.728,39.348,157.470
C04372=1045.622,256.613,395.129,171.726,39.345,157.469
C04373=1045.616,256.366,395.159,171.723,39.343,157.469
C04374=1045.609,256.117,395.188,171.721,39.341,157.468
C04375=1045.603,255.869,395.217,171.718,39.338,157.467
C04376=1045.596,255.621,395.247,171.715,39.335,157.467
C04377=1045.589,255.372,395.277,171.713,39.333,157.466
C04378=1045.583,255.124,395.306,171.709,39.330,157.465
C04379=1045.577,254.876,395.335,171.706,39.327,157.465
C04380=1045.570,254.628,395.365,171.704,39.325,157.464
C04381=1045.563,254.380,395.394,171.701,39.322,157.464
C04382=1045.557,254.132,395.423,171.699,39.320,157.463
C04383=1045.550,253.883,395.452,171.696,39.317,157.462
C04384=1045.543,253.635,395.481,171.693,39.315,157.462
C04385=1045.537,253.388,395.510,171.691,39.313,157.461
C04386=1045.530,253.139,395.540,171.688,39.310,157.460
C04387=1045.524,252.891,395.569,171.685,39.308,157.460
C04388=1045.517,252.642,395.598,171.682,39.305,157.459
C04389=1045.511,252.394,395.627,171.679,39.302,157.459
C04390=1045.504,252.146,395.656,171.677,39.300,157.458
C04391=1045.498,251.897,395.685,171.674,39.297,157.457
C04392=1045.492,251.649,395.714,171.672,39.294,157.457
C04393=1045.486,251.401,395.743,171.669,39.292,157.456
C04394=1045.478,251.153,395.772,171.666,39.289,157.455
C04395=1045.471,250.905,395.802,171.664,39.287,157.455
C04396=1045.465,250.657,395.831,171.661,39.284,157.454
C04397=1045.459,250.409,395.860,171.659,39.282,157.453
C04398=1045.452,250.160,395.890,171.656,39.279,157.453
C04399=1045.446,249.912,395.919,171.653,39.277,157.452
C04400=1045.440,249.664,395.948,171.650,39.274,157.452
C04401=1045.433,249.416,395.977,171.647,39.272,157.451
C04402=1045.426,249.140,396.009,171.645,39.269,157.450
C04403=1045.418,248.864,396.040,171.642,39.266,157.450
C04404=1045.411,248.588,396.072,171.639,39.263,157.449
C04405=1045.404,248.313,396.105,171.636,39.260,157.448
C04406=1045.398,248.065,396.134,171.633,39.258,157.448
C04407=1045.392,247.816,396.163,171.630,39.255,157.447
C04408=1045.385,247.568,396.192,171.628,39.253,157.446
C04409=1045.379,247.319,396.221,171.625,39.250,157.446
C04410=1045.373,247.071,396.250,171.623,39.248,157.445
C04411=1045.366,246.823,396.278,171.620,39.245,157.444
C04412=1045.360,246.575,396.307,171.617,39.243,157.444
C04413=1045.353,246.327,396.336,171.615,39.240,157.443
C04414=1045.347,246.079,396.365,171.612,39.237,157.443
C04415=1045.341,245.830,396.394,171.610,39.235,157.442
C04416=1045.334,245.581,396.423,171.607,39.232,157.441
C04417=1045.327,245.334,396.452,171.604,39.229,157.441
C04418=1045.321,245.085,396.481,171.602,39.227,157.440
C04419=1045.315,244.837,396.509,171.599,39.224,157.439
C04420=1045.308,244.589,396.537,171.597,39.222,157.439
C04421=1045.302,244.341,396.566,171.594,39.220,157.438
C04422=1045.295,244.092,396.594,171.591,39.217,157.438
C04423=1045.288,243.844,396.624,171.589,39.214,157.437
C04424=1045.282,243.595,396.653,171.586,39.212,157.436
C04425=1045.275,243.347,396.680,171.584,39.209,157.436
C04426=1045.269,243.099,396.709,171.582,39.206,157.435
C04427=1045.262,242.851,396.738,171.579,39.204,157.434
C04428=1045.256,242.602,396.766,171.577,39.202,157.434
C04429=1045.250,242.354,396.795,171.574,39.199,157.433
C04430=1045.243,242.106,396.824,171.572,39.197,157.433
C04431=1045.237,241.858,396.852,171.569,39.194,157.432
C04432=1045.230,241.610,396.880,171.567,39.191,157.431
C04433=1045.224,241.361,396.909,171.564,39.189,157.431
C04434=1045.217,241.113,396.937,171.561,39.186,157.430
C04435=1045.211,240.864,396.966,171.559,39.184,157.430
C04436=1045.204,240.616,396.994,171.556,39.182,157.429
C04437=1045.198,240.367,397.023,171.554,39.179,157.428
C04438=1045.191,240.119,397.051,171.551,39.177,157.428
C04439=1045.184,239.871,397.079,171.549,39.174,157.427
C04440=1045.178,239.622,397.107,171.546,39.171,157.426
C04441=1045.171,239.374,397.136,171.543,39.169,157.426
C04442=1045.164,239.126,397.163,171.541,39.167,157.425
C04443=1045.158,238.878,397.192,171.538,39.164,157.425
C04444=1045.151,238.629,397.220,171.536,39.162,157.424
C04445=1045.145,238.381,397.248,171.533,39.159,157.423
C04446=1045.138,238.133,397.277,171.532,39.156,157.423
C04447=1045.132,237.884,397.305,171.529,39.154,157.422
C04448=1045.125,237.636,397.333,171.526,39.151,157.422
C04449=1045.119,237.388,397.361,171.524,39.149,157.421
C04450=1045.112,237.139,397.389,171.521,39.147,157.421
C04451=1045.106,236.891,397.417,171.519,39.144,157.420
C04452=1045.099,236.643,397.445,171.516,39.141,157.419
C04453=1045.093,236.394,397.474,171.514,39.139,157.419
C04454=1045.086,236.146,397.501,171.511,39.136,157.418
C04455=1045.079,235.898,397.530,171.508,39.134,157.417
C04456=1045.073,235.649,397.558,171.506,39.132,157.417
C04457=1045.066,235.401,397.586,171.504,39.129,157.416
C04458=1045.059,235.119,397.617,171.501,39.127,157.416
C04459=1045.051,234.838,397.649,171.498,39.124,157.415
C04460=1045.044,234.556,397.681,171.495,39.121,157.414
C04461=1045.036,234.275,397.713,171.493,39.118,157.414
C04462=1045.030,234.027,397.741,171.490,39.115,157.413
C04463=1045.024,233.778,397.769,171.488,39.113,157.412
C04464=1045.018,233.530,397.797,171.485,39.110,157.412
C04465=1045.011,233.282,397.824,171.483,39.107,157.411
C04466=1045.004,233.033,397.852,171.481,39.105,157.411
C04467=1044.998,232.784,397.880,171.478,39.102,157.410
C04468=1044.991,232.537,397.909,171.476,39.100,157.409
C04469=1044.985,232.288,397.937,171.473,39.098,157.409
C04470=1044.978,232.040,397.964,171.471,39.095,157.408
C04471=1044.971,231.791,397.992,171.469,39.092,157.407
C04472=1044.965,231.543,398.020,171.467,39.090,157.407
C04473=1044.959,231.294,398.048,171.464,39.087,157.406
C04474=1044.952,231.046,398.075,171.461,39.085,157.406
C04475=1044.946,230.798,398.103,171.459,39.083,157.405
C04476=1044.939,230.549,398.131,171.456,39.080,157.404
C04477=1044.932,230.301,398.159,171.455,39.077,157.404
C04478=1044.926,230.053,398.186,171.452,39.075,157.403
C04479=1044.919,229.804,398.214,171.450,39.072,157.403
C04480=1044.912,229.556,398.242,171.447,39.070,157.402
C04481=1044.906,229.307,398.270,171.445,39.068,157.402
C04482=1044.900,229.059,398.298,171.442,39.065,157.401
C04483=1044.894,228.811,398.325,171.440,39.062,157.400
C04484=1044.887,228.562,398.353,171.438,39.060,157.400
C04485=1044.881,228.313,398.380,171.435,39.057,157.399
C04486=1044.874,228.065,398.408,171.433,39.055,157.398
C04487=1044.867,227.817,398.435,171.430,39.052,157.398
C04488=1044.860,227.568,398.463,171.429,39.049,157.397
C04489=1044.854,227.321,398.490,171.426,39.047,157.397
C04490=1044.847,227.072,398.518,171.423,39.045,157.396
C04491=1044.841,226.823,398.545,171.421,39.043,157.396
C04492=1044.834,226.575,398.572,171.418,39.040,157.395
C04493=1044.827,226.326,398.600,171.417,39.037,157.394
C04494=1044.821,226.078,398.628,171.414,39.035,157.394
C04495=1044.815,225.829,398.655,171.412,39.032,157.393
C04496=1044.807,225.581,398.682,171.409,39.030,157.393
C04497=1044.801,225.333,398.709,171.408,39.027,157.392
C04498=1044.794,225.084,398.737,171.405,39.025,157.391
C04499=1044.788,224.835,398.764,171.403,39.022,157.391
C04500=1044.782,224.588,398.792,171.400,39.020,157.390
C04501=1044.775,224.339,398.819,171.397,39.018,157.390
C04502=1044.768,224.091,398.847,171.396,39.015,157.389
C04503=1044.762,223.842,398.874,171.393,39.012,157.388
C04504=1044.755,223.594,398.901,171.391,39.010,157.388
C04505=1044.748,223.346,398.929,171.388,39.007,157.387
C04506=1044.742,223.097,398.956,171.387,39.005,157.387
C04507=1044.735,222.848,398.983,171.384,39.002,157.386
C04508=1044.730,222.600,399.010,171.382,39.000,157.385
C04509=1044.723,222.351,399.038,171.380,38.997,157.385
C04510=1044.716,222.103,399.065,171.377,38.994,157.384
C04511=1044.709,221.854,399.092,171.375,38.992,157.384
C04512=1044.703,221.606,399.119,171.372,38.990,157.383
C04513=1044.697,221.357,399.146,171.371,38.987,157.382
C04514=1044.689,221.068,399.178,171.368,38.984,157.382
C04515=1044.682,220.780,399.210,171.365,38.981,157.381
C04516=1044.675,220.491,399.241,171.363,38.978,157.380
C04517=1044.666,220.202,399.273,171.360,38.975,157.380
C04518=1044.660,219.953,399.300,171.358,38.973,157.379
C04519=1044.653,219.705,399.327,171.355,38.970,157.379
C04520=1044.647,219.456,399.354,171.354,38.967,157.378
C04521=1044.639,219.208,399.381,171.351,38.965,157.377
C04522=1044.633,218.959,399.408,171.349,38.963,157.377
C04523=1044.627,218.711,399.435,171.346,38.960,157.376
C04524=1044.620,218.463,399.462,171.344,38.957,157.376
C04525=1044.614,218.214,399.489,171.342,38.955,157.375
C04526=1044.607,217.966,399.516,171.339,38.953,157.374
C04527=1044.600,217.717,399.543,171.338,38.950,157.374
C04528=1044.594,217.469,399.570,171.335,38.948,157.373
C04529=1044.587,217.221,399.596,171.333,38.945,157.373
C04530=1044.581,216.972,399.623,171.331,38.942,157.372
C04531=1044.573,216.723,399.651,171.329,38.940,157.371
C04532=1044.568,216.475,399.677,171.326,38.938,157.371
C04533=1044.560,216.226,399.704,171.325,38.935,157.370
C04534=1044.554,215.978,399.731,171.322,38.932,157.370
C04535=1044.548,215.730,399.758,171.319,38.930,157.369
C04536=1044.541,215.481,399.784,171.318,38.927,157.369
C04537=1044.534,215.232,399.812,171.315,38.925,157.368
C04538=1044.528,214.984,399.838,171.313,38.922,157.367
C04539=1044.521,214.735,399.865,171.311,38.919,157.367
C04540=1044.515,214.487,399.891,171.309,38.917,157.366
C04541=1044.508,214.239,399.919,171.306,38.915,157.366
C04542=1044.502,213.990,399.946,171.305,38.912,157.365
C04543=1044.495,213.742,399.972,171.302,38.910,157.364
C04544=1044.489,213.493,399.999,171.301,38.907,157.364
C04545=1044.482,213.245,400.025,171.298,38.904,157.363
C04546=1044.476,212.996,400.053,171.295,38.902,157.363
C04547=1044.469,212.748,400.079,171.294,38.900,157.362
C04548=1044.463,212.499,400.106,171.291,38.897,157.361
C04549=1044.456,212.251,400.132,171.290,38.894,157.361
C04550=1044.450,212.002,400.159,171.287,38.891,157.360
C04551=1044.443,211.753,400.187,171.285,38.889,157.360
C04552=1044.437,211.505,400.213,171.283,38.887,157.359
C04553=1044.430,211.257,400.239,171.281,38.884,157.358
C04554=1044.424,211.008,400.266,171.278,38.881,157.358
C04555=1044.417,210.760,400.292,171.277,38.879,157.357
C04556=1044.410,210.511,400.318,171.274,38.876,157.357
C04557=1044.404,210.262,400.345,171.273,38.874,157.356
C04558=1044.397,210.014,400.371,171.270,38.871,157.356
C04559=1044.391,209.765,400.398,171.267,38.868,157.355
C04560=1044.384,209.517,400.424,171.266,38.866,157.354
C04561=1044.377,209.269,400.451,171.263,38.864,157.354
C04562=1044.371,209.019,400.478,171.262,38.861,157.353
C04563=1044.364,208.771,400.504,171.259,38.858,157.353
C04564=1044.357,208.523,400.530,171.258,38.856,157.352
C04565=1044.352,208.274,400.557,171.255,38.853,157.351
C04566=1044.344,208.026,400.583,171.253,38.851,157.351
C04567=1044.338,207.777,400.609,171.251,38.848,157.350
C04568=1044.331,207.529,400.636,171.249,38.845,157.350
C04569=1044.325,207.280,400.663,171.247,38.843,157.349
C04570=1044.318,206.997,400.693,171.244,38.840,157.348
C04571=1044.309,206.713,400.722,171.242,38.837,157.348
C04572=1044.302,206.430,400.753,171.239,38.834,157.347
C04573=1044.295,206.146,400.782,171.238,38.831,157.346
C04574=1044.269,205.095,400.889,170.974,38.730,157.319
C04575=1044.263,204.846,400.914,170.971,38.728,157.318
C04576=1044.257,204.597,400.939,170.968,38.726,157.318
C04577=1044.250,204.349,400.964,170.965,38.725,157.317
C04578=1044.244,204.100,400.989,170.962,38.723,157.317
C04579=1044.237,203.852,401.014,170.960,38.721,157.317
C04580=1044.232,203.604,401.039,170.957,38.719,157.316
C04581=1044.226,203.354,401.064,170.954,38.718,157.316
C04582=1044.220,203.106,401.089,170.951,38.715,157.315
C04583=1044.213,202.857,401.114,170.948,38.714,157.315
C04584=1044.207,202.608,401.140,170.946,38.712,157.314
C04585=1044.201,202.360,401.165,170.942,38.710,157.314
C04586=1044.196,202.111,401.189,170.940,38.709,157.314
C04587=1044.190,201.862,401.215,170.938,38.707,157.313
C04588=1044.183,201.614,401.240,170.934,38.705,157.313
C04589=1044.177,201.364,401.265,170.932,38.703,157.312
C04590=1044.170,201.116,401.289,170.929,38.702,157.312
C04591=1044.164,200.867,401.315,170.926,38.700,157.311
C04592=1044.159,200.619,401.339,170.923,38.698,157.311
C04593=1044.152,200.370,401.364,170.920,38.697,157.311
C04594=1044.146,200.121,401.388,170.918,38.695,157.310
C04595=1044.139,199.873,401.413,170.915,38.693,157.310
C04596=1044.133,199.623,401.438,170.912,38.692,157.309
C04597=1044.128,199.375,401.463,170.909,38.690,157.309
C04598=1044.121,199.127,401.487,170.907,38.688,157.309
C04599=1044.115,198.878,401.512,170.904,38.686,157.308
C04600=1044.108,198.629,401.536,170.901,38.685,157.308
C04601=1044.102,198.380,401.561,170.899,38.684,157.307
C04602=1044.096,198.132,401.585,170.895,38.682,157.307
C04603=1044.090,197.883,401.610,170.893,38.680,157.307
C04604=1044.084,197.634,401.635,170.890,38.679,157.306
C04605=1044.077,197.386,401.660,170.887,38.677,157.306
C04606=1044.072,197.137,401.684,170.885,38.675,157.305
C04607=1044.065,196.889,401.709,170.881,38.673,157.305
C04608=1044.059,196.639,401.733,170.879,38.672,157.305
C04609=1044.052,196.390,401.757,170.877,38.671,157.304
C04610=1044.046,196.142,401.782,170.873,38.669,157.304
C04611=1044.041,195.893,401.807,170.871,38.667,157.303
C04612=1044.034,195.645,401.832,170.868,38.665,157.303
C04613=1044.028,195.395,401.856,170.865,38.664,157.303
C04614=1044.022,195.147,401.880,170.863,38.662,157.302
C04615=1044.016,194.899,401.905,170.860,38.660,157.302
C04616=1044.009,194.650,401.929,170.857,38.659,157.301
C04617=1044.004,194.401,401.954,170.855,38.657,157.301
C04618=1043.997,194.153,401.978,170.852,38.656,157.301
C04619=1043.991,193.903,402.003,170.849,38.654,157.300
C04620=1043.985,193.655,402.027,170.847,38.652,157.300
C04621=1043.979,193.406,402.051,170.844,38.651,157.299
C04622=1043.973,193.157,402.077,170.841,38.649,157.299
C04623=1043.967,192.909,402.100,170.839,38.648,157.299
C04624=1043.961,192.660,402.125,170.836,38.646,157.298
C04625=1043.955,192.411,402.149,170.833,38.644,157.298
C04626=1043.948,192.163,402.174,170.831,38.643,157.297
C04627=1043.942,191.914,402.198,170.828,38.642,157.297
C04628=1043.936,191.665,402.222,170.825,38.640,157.297
C04629=1043.930,191.416,402.246,170.823,38.638,157.296
C04630=1043.924,191.168,402.271,170.820,38.636,157.296
C04631=1043.918,190.919,402.295,170.817,38.635,157.296
C04632=1043.912,190.670,402.320,170.815,38.633,157.295
C04633=1043.906,190.422,402.344,170.812,38.632,157.295
C04634=1043.900,190.172,402.368,170.809,38.630,157.294
C04635=1043.892,189.888,402.396,170.806,38.628,157.294
C04636=1043.886,189.604,402.423,170.804,38.627,157.294
C04637=1043.879,189.319,402.452,170.800,38.624,157.293
C04638=1043.872,189.034,402.479,170.798,38.623,157.293
C04639=1043.866,188.786,402.503,170.794,38.621,157.292
C04640=1043.860,188.537,402.528,170.792,38.620,157.292
C04641=1043.854,188.289,402.551,170.790,38.618,157.292
C04642=1043.848,188.039,402.576,170.786,38.616,157.291
C04643=1043.842,187.791,402.600,170.784,38.615,157.291
C04644=1043.836,187.542,402.624,170.782,38.613,157.290
C04645=1043.830,187.294,402.648,170.779,38.612,157.290
C04646=1043.825,187.044,402.672,170.776,38.610,157.290
C04647=1043.818,186.796,402.696,170.774,38.608,157.289
C04648=1043.813,186.547,402.721,170.771,38.607,157.289
C04649=1043.807,186.298,402.744,170.769,38.605,157.289
C04650=1043.801,186.049,402.769,170.766,38.604,157.288
C04651=1043.795,185.801,402.793,170.763,38.602,157.288
C04652=1043.789,185.552,402.817,170.761,38.601,157.287
C04653=1043.783,185.303,402.841,170.759,38.599,157.287
C04654=1043.777,185.055,402.865,170.755,38.597,157.287
C04655=1043.771,184.806,402.889,170.753,38.596,157.286
C04656=1043.765,184.557,402.913,170.751,38.595,157.286
C04657=1043.759,184.308,402.938,170.748,38.593,157.285
C04658=1043.753,184.060,402.961,170.746,38.591,157.285
C04659=1043.747,183.811,402.986,170.743,38.589,157.285
C04660=1043.741,183.562,403.009,170.740,38.588,157.284
C04661=1043.734,183.313,403.033,170.738,38.587,157.284
C04662=1043.728,183.064,403.056,170.735,38.585,157.284
C04663=1043.722,182.815,403.080,170.733,38.584,157.283
C04664=1043.716,182.567,403.103,170.730,38.583,157.283
C04665=1043.709,182.318,403.127,170.728,38.581,157.283
C04666=1043.703,182.069,403.151,170.725,38.580,157.282
C04667=1043.697,181.820,403.174,170.722,38.579,157.282
C04668=1043.691,181.571,403.198,170.720,38.577,157.282
C04669=1043.684,181.322,403.222,170.718,38.576,157.281
C04670=1043.678,181.074,403.244,170.715,38.575,157.281
C04671=1043.671,180.825,403.268,170.712,38.573,157.281
C04672=1043.665,180.577,403.292,170.710,38.572,157.280
C04673=1043.660,180.328,403.315,170.708,38.570,157.280
C04674=1043.653,180.079,403.339,170.704,38.569,157.280
C04675=1043.647,179.830,403.362,170.702,38.568,157.279
C04676=1043.641,179.581,403.386,170.700,38.566,157.279
C04677=1043.635,179.332,403.409,170.698,38.565,157.279
C04678=1043.628,179.083,403.433,170.694,38.563,157.278
C04679=1043.622,178.835,403.457,170.692,38.562,157.278
C04680=1043.616,178.585,403.480,170.690,38.561,157.278
C04681=1043.610,178.337,403.504,170.687,38.559,157.277
C04682=1043.603,178.088,403.526,170.684,38.558,157.277
C04683=1043.597,177.839,403.550,170.682,38.556,157.277
C04684=1043.591,177.590,403.573,170.680,38.555,157.276
C04685=1043.584,177.341,403.597,170.677,38.554,157.276
C04686=1043.579,177.092,403.620,170.675,38.552,157.276
C04687=1043.572,176.844,403.644,170.672,38.551,157.275
C04688=1043.566,176.595,403.667,170.669,38.550,157.275
C04689=1043.560,176.346,403.691,170.667,38.548,157.275
C04690=1043.554,176.097,403.714,170.665,38.547,157.274
C04691=1043.547,175.849,403.737,170.663,38.546,157.274
C04692=1043.541,175.600,403.760,170.659,38.545,157.274
C04693=1043.536,175.351,403.783,170.657,38.543,157.273
C04694=1043.529,175.102,403.807,170.655,38.542,157.273
C04695=1043.523,174.853,403.830,170.652,38.540,157.273
C04696=1043.517,174.605,403.854,170.650,38.539,157.272
C04697=1043.511,174.355,403.877,170.647,38.538,157.272
C04698=1043.505,174.106,403.900,170.645,38.537,157.272
C04699=1043.497,173.822,403.927,170.642,38.535,157.271
C04700=1043.491,173.537,403.953,170.639,38.533,157.271
C04701=1043.483,173.252,403.980,170.637,38.532,157.271
C04702=1043.477,172.967,404.006,170.633,38.530,157.270
C04703=1043.471,172.718,404.029,170.631,38.529,157.270
C04704=1043.465,172.470,404.053,170.629,38.527,157.270
C04705=1043.459,172.221,404.076,170.627,38.526,157.269
C04706=1043.452,171.972,404.098,170.624,38.524,157.269
C04707=1043.446,171.723,404.121,170.622,38.523,157.269
C04708=1043.440,171.474,404.145,170.619,38.522,157.268
C04709=1043.435,171.226,404.168,170.616,38.520,157.268
C04710=1043.428,170.976,404.191,170.614,38.519,157.268
C04711=1043.422,170.728,404.215,170.612,38.518,157.267
C04712=1043.416,170.479,404.237,170.610,38.516,157.267
C04713=1043.410,170.230,404.260,170.607,38.515,157.267
C04714=1043.404,169.981,404.284,170.605,38.514,157.266
C04715=1043.398,169.732,404.307,170.602,38.512,157.266
C04716=1043.392,169.483,404.330,170.599,38.511,157.266
C04717=1043.386,169.235,404.353,170.597,38.510,157.265
C04718=1043.380,168.986,404.376,170.595,38.508,157.265
C04719=1043.374,168.737,404.398,170.593,38.507,157.265
C04720=1043.368,168.487,404.422,170.590,38.506,157.264
C04721=1043.362,168.239,404.445,170.588,38.504,157.264
C04722=1043.356,167.990,404.468,170.586,38.503,157.264
C04723=1043.350,167.741,404.491,170.584,38.502,157.264
C04724=1043.344,167.493,404.514,170.580,38.500,157.263
C04725=1043.338,167.244,404.537,170.578,38.499,157.263
C04726=1043.332,166.994,404.560,170.576,38.498,157.263
C04727=1043.326,166.745,404.583,170.573,38.496,157.262
C04728=1043.320,166.497,404.606,170.571,38.495,157.262
C04729=1043.314,166.248,404.629,170.569,38.494,157.262
C04730=1043.308,165.999,404.651,170.567,38.492,157.261
C04731=1043.302,165.750,404.674,170.564,38.491,157.261
C04732=1043.296,165.501,404.697,170.562,38.490,157.261
C04733=1043.290,165.253,404.721,170.560,38.488,157.260
C04734=1043.285,165.004,404.744,170.558,38.487,157.260
C04735=1043.278,164.755,404.766,170.554,38.486,157.260
C04736=1043.272,164.506,404.789,170.552,38.484,157.259
C04737=1043.266,164.257,404.812,170.550,38.483,157.259
C04738=1043.260,164.008,404.835,170.547,38.482,157.259
C04739=1043.255,163.759,404.858,170.545,38.480,157.258
C04740=1043.248,163.511,404.880,170.543,38.479,157.258
C04741=1043.243,163.261,404.903,170.541,38.478,157.258
C04742=1043.237,163.012,404.926,170.538,38.476,157.257
C04743=1043.231,162.763,404.949,170.536,38.475,157.257
C04744=1043.225,162.515,404.971,170.534,38.474,157.257
C04745=1043.219,162.266,404.994,170.531,38.472,157.256
C04746=1043.213,162.017,405.017,170.529,38.471,157.256
C04747=1043.208,161.768,405.040,170.527,38.470,157.256
C04748=1043.202,161.519,405.063,170.525,38.468,157.255
C04749=1043.195,161.271,405.085,170.522,38.467,157.255
C04750=1043.190,161.022,405.108,170.520,38.466,157.255
C04751=1043.184,160.773,405.131,170.518,38.464,157.255
C04752=1043.179,160.523,405.153,170.516,38.463,157.254
C04753=1043.172,160.275,405.176,170.513,38.462,157.254
C04754=1043.166,160.026,405.199,170.511,38.461,157.254
C04755=1043.160,159.777,405.221,170.508,38.460,157.253
C04756=1043.154,159.528,405.244,170.506,38.458,157.253
C04757=1043.148,159.279,405.265,170.503,38.457,157.253
C04758=1043.142,159.030,405.288,170.501,38.456,157.252
C04759=1043.135,158.781,405.311,170.499,38.454,157.252
C04760=1043.129,158.532,405.333,170.497,38.453,157.252
C04761=1043.123,158.283,405.356,170.494,38.452,157.252
C04762=1043.117,158.034,405.378,170.492,38.451,157.251
C04763=1043.110,157.749,405.403,170.490,38.449,157.251
C04764=1043.103,157.464,405.429,170.487,38.448,157.251
C04765=1043.096,157.178,405.454,170.484,38.447,157.250
C04766=1043.089,156.893,405.481,170.482,38.445,157.250
C04767=1043.083,156.644,405.502,170.480,38.444,157.250
C04768=1043.077,156.396,405.525,170.478,38.443,157.249
C04769=1043.071,156.146,405.547,170.475,38.442,157.249
C04770=1043.065,155.897,405.569,170.473,38.441,157.249
C04771=1043.059,155.649,405.592,170.470,38.440,157.249
C04772=1043.053,155.399,405.614,170.468,38.438,157.248
C04773=1043.047,155.151,405.636,170.465,38.437,157.248
C04774=1043.040,154.902,405.658,170.463,38.436,157.248
C04775=1043.035,154.653,405.681,170.461,38.434,157.247
C04776=1043.029,154.403,405.702,170.459,38.433,157.247
C04777=1043.022,154.155,405.725,170.456,38.432,157.247
C04778=1043.017,153.905,405.747,170.454,38.431,157.247
C04779=1043.010,153.657,405.769,170.452,38.430,157.246
C04780=1043.004,153.408,405.791,170.450,38.429,157.246
C04781=1042.998,153.159,405.813,170.447,38.427,157.246
C04782=1042.991,152.910,405.835,170.445,38.426,157.245
C04783=1042.986,152.661,405.858,170.443,38.425,157.245
C04784=1042.980,152.412,405.880,170.441,38.424,157.245
C04785=1042.973,152.163,405.902,170.438,38.423,157.245
C04786=1042.967,151.914,405.924,170.436,38.422,157.244
C04787=1042.962,151.666,405.946,170.434,38.421,157.244
C04788=1042.956,151.417,405.968,170.432,38.419,157.244
C04789=1042.949,151.168,405.990,170.430,38.418,157.244
C04790=1042.943,150.919,406.012,170.427,38.417,157.243
C04791=1042.937,150.670,406.033,170.425,38.416,157.243
C04792=1042.931,150.421,406.056,170.423,38.415,157.243
C04793=1042.925,150.171,406.078,170.421,38.414,157.242
C04794=1042.919,149.922,406.100,170.418,38.413,157.242
C04795=1042.912,149.674,406.122,170.416,38.411,157.242
C04796=1042.906,149.424,406.144,170.414,38.410,157.242
C04797=1042.901,149.176,406.165,170.412,38.409,157.241
C04798=1042.895,148.927,406.188,170.409,38.408,157.241
C04799=1042.889,148.678,406.209,170.407,38.407,157.241
C04800=1042.882,148.429,406.231,170.405,38.406,157.241
C04801=1042.876,148.180,406.253,170.403,38.405,157.240
C04802=1042.870,147.931,406.275,170.401,38.403,157.240
C04803=1042.864,147.682,406.297,170.398,38.402,157.240
C04804=1042.858,147.432,406.318,170.396,38.401,157.239
C04805=1042.852,147.185,406.340,170.394,38.400,157.239
C04806=1042.846,146.935,406.363,170.392,38.399,157.239
C04807=1042.839,146.686,406.384,170.389,38.398,157.239
C04808=1042.833,146.437,406.405,170.387,38.397,157.238
C04809=1042.827,146.188,406.428,170.385,38.395,157.238
C04810=1042.821,145.939,406.449,170.383,38.394,157.238
C04811=1042.814,145.690,406.471,170.380,38.393,157.238
C04812=1042.809,145.441,406.492,170.378,38.392,157.237
C04813=1042.803,145.192,406.514,170.376,38.391,157.237
C04814=1042.796,144.943,406.535,170.374,38.390,157.237
C04815=1042.790,144.694,406.558,170.372,38.389,157.237
C04816=1042.784,144.445,406.579,170.370,38.388,157.236
C04817=1042.778,144.196,406.601,170.368,38.387,157.236
C04818=1042.772,143.947,406.622,170.366,38.386,157.236
C04819=1042.766,143.698,406.644,170.364,38.384,157.235
C04820=1042.760,143.449,406.666,170.362,38.383,157.235
C04821=1042.754,143.200,406.687,170.359,38.382,157.235
C04822=1042.747,142.951,406.709,170.357,38.381,157.235
C04823=1042.742,142.702,406.730,170.355,38.380,157.234
C04824=1042.736,142.453,406.752,170.353,38.379,157.234
C04825=1042.730,142.204,406.773,170.350,38.378,157.234
C04826=1042.722,141.955,406.795,170.348,38.377,157.234
C04827=1042.716,141.670,406.819,170.346,38.376,157.233
C04828=1042.709,141.384,406.845,170.343,38.374,157.233
C04829=1042.703,141.098,406.869,170.340,38.373,157.233
C04830=1042.695,140.813,406.894,170.338,38.372,157.232
C04831=1042.689,140.564,406.915,170.336,38.371,157.232
C04832=1042.683,140.315,406.937,170.334,38.370,157.232
C04833=1042.677,140.066,406.958,170.332,38.368,157.232
C04834=1042.671,139.817,406.980,170.329,38.367,157.231
C04835=1042.665,139.567,407.001,170.327,38.366,157.231
C04836=1042.659,139.319,407.023,170.325,38.366,157.231
C04837=1042.653,139.070,407.044,170.323,38.364,157.231
C04838=1042.646,138.820,407.065,170.321,38.363,157.230
C04839=1042.641,138.572,407.086,170.319,38.362,157.230
C04840=1042.634,138.323,407.108,170.317,38.361,157.230
C04841=1042.628,138.073,407.129,170.315,38.360,157.230
C04842=1042.621,137.824,407.150,170.313,38.359,157.229
C04843=1042.616,137.576,407.172,170.310,38.358,157.229
C04844=1042.610,137.327,407.193,170.308,38.357,157.229
C04845=1042.604,137.078,407.215,170.306,38.356,157.229
C04846=1042.597,136.828,407.235,170.304,38.355,157.228
C04847=1042.591,136.579,407.256,170.302,38.353,157.228
C04848=1042.585,136.330,407.278,170.299,38.353,157.228
C04849=1042.578,136.081,407.299,170.297,38.352,157.228
C04850=1042.573,135.833,407.320,170.295,38.351,157.227
C04851=1042.567,135.583,407.341,170.293,38.349,157.227
C04852=1042.560,135.334,407.362,170.291,38.348,157.227
C04853=1042.554,135.086,407.384,170.289,38.348,157.227
C04854=1042.548,134.836,407.405,170.287,38.347,157.226
C04855=1042.542,134.587,407.427,170.285,38.345,157.226
C04856=1042.536,134.338,407.447,170.283,38.344,157.226
C04857=1042.530,134.089,407.468,170.280,38.343,157.226
C04858=1042.524,133.840,407.490,170.278,38.342,157.225
C04859=1042.518,133.591,407.510,170.276,38.341,157.225
C04860=1042.512,133.342,407.532,170.274,38.340,157.225
C04861=1042.505,133.093,407.553,170.272,38.339,157.225
C04862=1042.499,132.845,407.574,170.269,38.338,157.224
C04863=1042.493,132.595,407.595,170.267,38.337,157.224
C04864=1042.487,132.346,407.617,170.266,38.336,157.224
C04865=1042.481,132.097,407.637,170.264,38.335,157.224
C04866=1042.475,131.848,407.658,170.262,38.334,157.223
C04867=1042.469,131.599,407.679,170.259,38.333,157.223
C04868=1042.463,131.350,407.700,170.257,38.332,157.223
C04869=1042.457,131.100,407.721,170.255,38.331,157.223
C04870=1042.450,130.852,407.742,170.253,38.330,157.222
C04871=1042.445,130.602,407.763,170.251,38.329,157.222
C04872=1042.438,130.353,407.784,170.249,38.328,157.222
C04873=1042.432,130.105,407.804,170.246,38.327,157.222
C04874=1042.425,129.855,407.826,170.244,38.326,157.222
C04875=1042.419,129.606,407.846,170.243,38.325,157.221
C04876=1042.413,129.358,407.867,170.241,38.324,157.221
C04877=1042.407,129.108,407.888,170.239,38.323,157.221
C04878=1042.400,128.859,407.909,170.236,38.322,157.221
C04879=1042.394,128.610,407.929,170.234,38.321,157.220
C04880=1042.388,128.361,407.950,170.232,38.320,157.220
C04881=1042.382,128.112,407.970,170.230,38.320,157.220
C04882=1042.375,127.863,407.992,170.228,38.318,157.220
C04883=1042.369,127.613,408.012,170.225,38.317,157.219
C04884=1042.363,127.365,408.033,170.223,38.317,157.219
C04885=1042.357,127.115,408.054,170.221,38.316,157.219
C04886=1042.350,126.867,408.074,170.220,38.314,157.219
C04887=1042.344,126.618,408.095,170.218,38.314,157.219
C04888=1042.338,126.368,408.116,170.215,38.313,157.218
C04889=1042.332,126.120,408.136,170.213,38.312,157.218
C04890=1042.325,125.870,408.157,170.211,38.311,157.218
C04891=1042.318,125.585,408.180,170.209,38.310,157.218
C04892=1042.310,125.299,408.204,170.207,38.309,157.217
C04893=1042.304,125.013,408.228,170.204,38.307,157.217
C04894=1042.298,124.727,408.251,170.201,38.306,157.217
C04895=1042.291,124.478,408.272,170.199,38.305,157.217
C04896=1042.284,124.229,408.293,170.198,38.304,157.216
C04897=1042.279,123.979,408.313,170.196,38.303,157.216
C04898=1042.272,123.731,408.334,170.193,38.302,157.216
C04899=1042.266,123.482,408.354,170.191,38.301,157.216
C04900=1042.260,123.232,408.375,170.189,38.301,157.215
C04901=1042.254,122.984,408.396,170.187,38.299,157.215
C04902=1042.247,122.734,408.416,170.185,38.298,157.215
C04903=1042.242,122.485,408.437,170.184,38.298,157.215
C04904=1042.235,122.236,408.458,170.181,38.297,157.215
C04905=1042.229,121.987,408.478,170.179,38.295,157.214
C04906=1042.222,121.738,408.498,170.177,38.295,157.214
C04907=1042.217,121.489,408.519,170.175,38.294,157.214
C04908=1042.210,121.240,408.540,170.172,38.293,157.214
C04909=1042.204,120.991,408.560,170.170,38.291,157.213
C04910=1042.199,120.742,408.580,170.169,38.291,157.213
C04911=1042.192,120.492,408.601,170.167,38.290,157.213
C04912=1042.186,120.244,408.621,170.165,38.288,157.213
C04913=1042.180,119.994,408.642,170.163,38.288,157.212
C04914=1042.174,119.746,408.662,170.160,38.287,157.212
C04915=1042.168,119.496,408.682,170.158,38.286,157.212
C04916=1042.162,119.247,408.702,170.156,38.285,157.212
C04917=1042.155,118.998,408.724,170.155,38.284,157.212
C04918=1042.149,118.749,408.744,170.153,38.283,157.211
C04919=1042.143,118.500,408.764,170.150,38.282,157.211
C04920=1042.138,118.251,408.785,170.148,38.281,157.211
C04921=1042.132,118.002,408.805,170.146,38.280,157.211
C04922=1042.125,117.752,408.825,170.144,38.279,157.210
C04923=1042.119,117.504,408.846,170.143,38.278,157.210
C04924=1042.113,117.255,408.866,170.140,38.277,157.210
C04925=1042.107,117.005,408.887,170.138,38.276,157.210
C04926=1042.101,116.757,408.907,170.136,38.275,157.209
C04927=1042.095,116.507,408.928,170.134,38.274,157.209
C04928=1042.089,116.258,408.948,170.132,38.273,157.209
C04929=1042.083,116.009,408.968,170.130,38.272,157.209
C04930=1042.076,115.760,408.988,170.128,38.271,157.208
C04931=1042.071,115.511,409.009,170.126,38.270,157.208
C04932=1042.065,115.262,409.029,170.124,38.269,157.208
C04933=1042.058,115.013,409.049,170.122,38.268,157.208
C04934=1042.053,114.764,409.070,170.121,38.267,157.208
C04935=1042.047,114.515,409.090,170.118,38.266,157.207
C04936=1042.040,114.265,409.110,170.116,38.265,157.207
C04937=1042.034,114.017,409.130,170.114,38.264,157.207
C04938=1042.029,113.767,409.151,170.112,38.263,157.207
C04939=1042.023,113.518,409.171,170.111,38.262,157.206
C04940=1042.017,113.269,409.191,170.108,38.261,157.206
C04941=1042.010,113.020,409.211,170.106,38.260,157.206
C04942=1042.004,112.771,409.231,170.104,38.259,157.206
C04943=1041.998,112.522,409.251,170.102,38.258,157.205
C04944=1041.991,112.272,409.272,170.100,38.257,157.205
C04945=1041.986,112.023,409.291,170.098,38.256,157.205
C04946=1041.980,111.774,409.311,170.096,38.256,157.205
C04947=1041.973,111.525,409.331,170.094,38.254,157.205
C04948=1041.967,111.276,409.351,170.092,38.253,157.204
C04949=1041.961,111.027,409.371,170.090,38.253,157.204
C04950=1041.955,110.777,409.391,170.088,38.251,157.204
C04951=1041.949,110.529,409.411,170.086,38.251,157.204
C04952=1041.943,110.280,409.431,170.084,38.250,157.204
C04953=1041.936,110.030,409.451,170.082,38.249,157.203
C04954=1041.930,109.781,409.470,170.080,38.248,157.203
C04955=1041.923,109.495,409.493,170.078,38.247,157.203
C04956=1041.916,109.208,409.517,170.075,38.246,157.203
C04957=1041.908,108.923,409.539,170.073,38.245,157.202
C04958=1041.901,108.637,409.562,170.071,38.244,157.202
C04959=1041.895,108.388,409.582,170.069,38.243,157.202
C04960=1041.888,108.139,409.601,170.067,38.242,157.202
C04961=1041.882,107.890,409.621,170.064,38.241,157.202
C04962=1041.876,107.641,409.641,170.062,38.241,157.201
C04963=1041.870,107.391,409.661,170.060,38.239,157.201
C04964=1041.864,107.142,409.681,170.059,38.239,157.201
C04965=1041.858,106.893,409.701,170.057,38.238,157.201
C04966=1041.851,106.644,409.720,170.055,38.237,157.201
C04967=1041.845,106.395,409.740,170.052,38.236,157.200
C04968=1041.839,106.146,409.760,170.050,38.235,157.200
C04969=1041.833,105.896,409.779,170.049,38.234,157.200
C04970=1041.827,105.647,409.799,170.047,38.233,157.200
C04971=1041.821,105.398,409.819,170.045,38.232,157.199
C04972=1041.814,105.150,409.839,170.043,38.231,157.199
C04973=1041.808,104.900,409.858,170.040,38.231,157.199
C04974=1041.802,104.651,409.878,170.039,38.230,157.199
C04975=1041.796,104.401,409.898,170.037,38.228,157.199
C04976=1041.790,104.152,409.918,170.035,38.228,157.198
C04977=1041.783,103.904,409.937,170.033,38.227,157.198
C04978=1041.777,103.654,409.957,170.031,38.226,157.198
C04979=1041.771,103.405,409.976,170.028,38.225,157.198
C04980=1041.765,103.156,409.996,170.027,38.224,157.198
C04981=1041.759,102.907,410.016,170.025,38.223,157.197
C04982=1041.753,102.658,410.036,170.023,38.222,157.197
C04983=1041.746,102.408,410.055,170.021,38.221,157.197
C04984=1041.740,102.159,410.075,170.018,38.220,157.197
C04985=1041.734,101.911,410.095,170.017,38.220,157.196
C04986=1041.728,101.661,410.114,170.015,38.219,157.196
C04987=1041.722,101.412,410.134,170.013,38.217,157.196
C04988=1041.715,101.162,410.153,170.011,38.217,157.196
C04989=1041.709,100.914,410.173,170.010,38.216,157.196
C04990=1041.704,100.664,410.192,170.007,38.215,157.195
C04991=1041.698,100.415,410.212,170.005,38.214,157.195
C04992=1041.691,100.166,410.231,170.003,38.213,157.195
C04993=1041.685,99.917,410.251,170.001,38.212,157.195
C04994=1041.678,99.668,410.270,169.999,38.212,157.195
C04995=1041.672,99.419,410.290,169.998,38.210,157.194
C04996=1041.667,99.169,410.309,169.995,38.210,157.194
C04997=1041.660,98.921,410.328,169.993,38.209,157.194
C04998=1041.654,98.671,410.348,169.991,38.208,157.194
C04999=1041.647,98.422,410.366,169.989,38.207,157.193
C05000=1041.641,98.173,410.386,169.988,38.206,157.193
C05001=1041.635,97.924,410.405,169.986,38.205,157.193
C05002=1041.629,97.675,410.425,169.983,38.205,157.193
C05003=1041.622,97.425,410.444,169.981,38.204,157.193
C05004=1041.616,97.176,410.463,169.979,38.203,157.193
C05005=1041.609,96.927,410.483,169.978,38.202,157.192
C05006=1041.604,96.678,410.502,169.976,38.201,157.192
C05007=1041.598,96.428,410.521,169.974,38.201,157.192
C05008=1041.591,96.180,410.540,169.971,38.200,157.192
C05009=1041.586,95.930,410.560,169.969,38.199,157.192
C05010=1041.578,95.680,410.579,169.968,38.198,157.191
C05011=1041.572,95.432,410.599,169.966,38.197,157.191
C05012=1041.566,95.183,410.617,169.964,38.196,157.191
C05013=1041.560,94.933,410.637,169.962,38.195,157.191
C05014=1041.554,94.685,410.656,169.959,38.194,157.191
C05015=1041.548,94.435,410.675,169.958,38.194,157.190
C05016=1041.542,94.186,410.694,169.956,38.193,157.190
C05017=1041.536,93.937,410.714,169.954,38.192,157.190
C05018=1041.529,93.687,410.733,169.952,38.191,157.190
C05019=1041.522,93.402,410.754,169.950,38.190,157.189
C05020=1041.515,93.116,410.777,169.947,38.189,157.189
C05021=1041.508,92.829,410.799,169.945,38.188,157.189
C05022=1041.501,92.544,410.821,169.943,38.187,157.189
C05023=1041.494,92.295,410.840,169.941,38.186,157.189
C05024=1041.489,92.045,410.859,169.939,38.185,157.188
C05025=1041.482,91.796,410.877,169.938,38.184,157.188
C05026=1041.476,91.547,410.897,169.935,38.183,157.188
C05027=1041.470,91.298,410.916,169.933,38.183,157.188
C05028=1041.464,91.049,410.935,169.931,38.182,157.188
C05029=1041.457,90.799,410.954,169.930,38.181,157.187
C05030=1041.451,90.549,410.974,169.928,38.180,157.187
C05031=1041.446,90.300,410.993,169.926,38.179,157.187
C05032=1041.439,90.052,411.012,169.923,38.178,157.187
C05033=1041.433,89.802,411.031,169.921,38.178,157.187
C05034=1041.426,89.553,411.049,169.920,38.176,157.186
C05035=1041.420,89.304,411.069,169.918,38.176,157.186
C05036=1041.414,89.055,411.087,169.916,38.175,157.186
C05037=1041.408,88.806,411.106,169.914,38.174,157.186
C05038=1041.401,88.556,411.125,169.912,38.173,157.186
C05039=1041.395,88.307,411.144,169.910,38.173,157.185
C05040=1041.389,88.058,411.163,169.908,38.172,157.185
C05041=1041.383,87.809,411.181,169.906,38.171,157.185
C05042=1041.376,87.560,411.200,169.904,38.170,157.185
C05043=1041.370,87.310,411.219,169.902,38.169,157.185
C05044=1041.363,87.060,411.238,169.901,38.169,157.185
C05045=1041.357,86.811,411.257,169.898,38.168,157.184
C05046=1041.351,86.562,411.275,169.896,38.167,157.184
C05047=1041.344,86.313,411.294,169.894,38.166,157.184
C05048=1041.338,86.064,411.313,169.892,38.165,157.184
C05049=1041.332,85.814,411.332,169.891,38.165,157.184
C05050=1041.326,85.565,411.351,169.889,38.164,157.183
C05051=1041.319,85.316,411.369,169.887,38.163,157.183
C05052=1041.313,85.067,411.389,169.884,38.162,157.183
C05053=1041.307,84.818,411.407,169.882,38.161,157.183
C05054=1041.301,84.569,411.426,169.881,38.161,157.183
C05055=1041.294,84.319,411.444,169.879,38.160,157.182
C05056=1041.288,84.070,411.463,169.877,38.159,157.182
C05057=1041.282,83.821,411.482,169.875,38.158,157.182
C05058=1041.276,83.572,411.501,169.872,38.157,157.182
C05059=1041.269,83.323,411.520,169.871,38.156,157.182
C05060=1041.263,83.073,411.538,169.869,38.156,157.181
C05061=1041.257,82.824,411.556,169.867,38.155,157.181
C05062=1041.252,82.575,411.575,169.865,38.154,157.181
C05063=1041.245,82.326,411.594,169.864,38.153,157.181
C05064=1041.239,82.077,411.612,169.861,38.152,157.181
C05065=1041.232,81.828,411.631,169.859,38.152,157.180
C05066=1041.226,81.579,411.650,169.857,38.150,157.180
C05067=1041.220,81.329,411.669,169.855,38.150,157.180
C05068=1041.214,81.079,411.687,169.854,38.149,157.180
C05069=1041.208,80.830,411.706,169.852,38.148,157.180
C05070=1041.201,80.581,411.724,169.850,38.147,157.180
C05071=1041.195,80.332,411.743,169.847,38.146,157.179
C05072=1041.189,80.083,411.762,169.846,38.146,157.179
C05073=1041.183,79.833,411.781,169.844,38.145,157.179
C05074=1041.177,79.584,411.799,169.842,38.144,157.179
C05075=1041.171,79.335,411.817,169.840,38.143,157.178
C05076=1041.164,79.086,411.836,169.838,38.142,157.178
C05077=1041.158,78.837,411.854,169.836,38.141,157.178
C05078=1041.153,78.587,411.873,169.834,38.140,157.178
C05079=1041.146,78.338,411.891,169.832,38.140,157.178
C05080=1041.140,78.089,411.910,169.830,38.139,157.178
C05081=1041.133,77.840,411.929,169.829,38.138,157.177
C05082=1041.127,77.590,411.947,169.827,38.137,157.177
C05083=1041.121,77.367,411.963,169.824,38.136,157.177
C05084=1041.116,77.145,411.980,169.823,38.136,157.177
C05085=1041.110,76.921,411.996,169.821,38.135,157.177
C05086=1041.105,76.699,412.013,169.819,38.135,157.177
C05087=1041.099,76.475,412.029,169.818,38.134,157.176
C05088=1041.093,76.253,412.045,169.816,38.133,157.176
C05089=1041.088,76.030,412.062,169.815,38.132,157.176
C05090=1041.082,75.807,412.078,169.813,38.132,157.176
C05091=1041.076,75.558,412.097,169.810,38.131,157.176
C05092=1041.070,75.308,412.115,169.808,38.130,157.175
C05093=1041.063,75.060,412.132,169.807,38.129,157.175
C05094=1041.057,74.811,412.151,169.805,38.128,157.175
C05095=1041.051,74.561,412.169,169.803,38.128,157.175
C05096=1041.044,74.312,412.188,169.801,38.127,157.175
C05097=1041.038,74.062,412.205,169.798,38.126,157.175
C05098=1041.032,73.813,412.224,169.797,38.125,157.174
C05099=1041.025,73.564,412.243,169.795,38.125,157.174
C05100=1041.020,73.315,412.260,169.793,38.124,157.174
C05101=1041.013,73.066,412.279,169.791,38.123,157.174
C05102=1041.007,72.816,412.297,169.789,38.123,157.174
C05103=1041.001,72.567,412.316,169.788,38.121,157.173
C05104=1040.995,72.317,412.333,169.786,38.121,157.173
C05105=1040.988,72.068,412.352,169.783,38.120,157.173
C05106=1040.982,71.819,412.369,169.781,38.119,157.173
C05107=1040.976,71.570,412.388,169.779,38.119,157.173
C05108=1040.969,71.321,412.406,169.778,38.117,157.173
C05109=1040.963,71.071,412.424,169.776,38.117,157.172
C05110=1040.957,70.822,412.442,169.774,38.116,157.172
C05111=1040.948,70.483,412.467,169.771,38.115,157.172
C05112=1040.940,70.145,412.492,169.768,38.114,157.172
C05113=1040.932,69.806,412.516,169.766,38.113,157.171
C05114=1040.923,69.467,412.541,169.763,38.112,157.171
C05115=1040.917,69.218,412.558,169.762,38.111,157.171
C05116=1040.911,68.969,412.577,169.760,38.110,157.171
C05117=1040.905,68.719,412.595,169.757,38.109,157.171
C05118=1040.898,68.470,412.612,169.755,38.109,157.170
C05119=1040.891,68.220,412.631,169.753,38.108,157.170
C05120=1040.886,67.971,412.649,169.752,38.107,157.170
C05121=1040.880,67.722,412.666,169.750,38.106,157.170
C05122=1040.872,67.473,412.685,169.748,38.106,157.170
C05123=1040.866,67.223,412.702,169.745,38.105,157.170
C05124=1040.861,66.974,412.720,169.743,38.104,157.169
C05125=1040.854,66.725,412.739,169.742,38.103,157.169
C05126=1040.847,66.476,412.756,169.740,38.103,157.169
C05127=1040.841,66.226,412.774,169.738,38.102,157.169
C05128=1040.836,65.977,412.792,169.736,38.101,157.169
C05129=1040.829,65.728,412.810,169.734,38.101,157.169
C05130=1040.823,65.478,412.827,169.732,38.099,157.168
C05131=1040.816,65.229,412.846,169.730,38.099,157.168
C05132=1040.810,64.980,412.863,169.728,38.098,157.168
C05133=1040.804,64.731,412.881,169.726,38.097,157.168
C05134=1040.798,64.481,412.899,169.724,38.097,157.168
C05135=1040.790,64.232,412.917,169.723,38.096,157.167
C05136=1040.785,63.983,412.935,169.721,38.095,157.167
C05137=1040.779,63.733,412.953,169.718,38.094,157.167
C05138=1040.772,63.484,412.970,169.716,38.094,157.167
C05139=1040.765,63.234,412.987,169.714,38.093,157.167
C05140=1040.759,62.986,413.005,169.712,38.093,157.167
C05141=1040.752,62.737,413.023,169.711,38.092,157.167
C05142=1040.746,62.487,413.041,169.709,38.091,157.166
C05143=1040.739,62.237,413.058,169.707,38.090,157.166
C05144=1040.733,61.989,413.075,169.705,38.090,157.166
C05145=1040.727,61.739,413.093,169.703,38.089,157.166
C05146=1040.720,61.489,413.110,169.700,38.089,157.166
C05147=1040.713,61.204,413.130,169.698,38.087,157.165
C05148=1040.706,60.917,413.151,169.696,38.087,157.165
C05149=1040.698,60.630,413.171,169.694,38.086,157.165
C05150=1040.691,60.345,413.192,169.692,38.085,157.165
C05151=1040.684,60.096,413.209,169.690,38.085,157.165
C05152=1040.678,59.846,413.227,169.688,38.084,157.165
C05153=1040.672,59.597,413.244,169.686,38.083,157.164
C05154=1040.666,59.347,413.262,169.684,38.083,157.164
C05155=1040.659,59.098,413.279,169.682,38.082,157.164
C05156=1040.652,58.849,413.296,169.680,38.081,157.164
C05157=1040.646,58.599,413.314,169.678,38.081,157.164
C05158=1040.639,58.350,413.331,169.676,38.080,157.164
C05159=1040.634,58.101,413.349,169.675,38.079,157.164
C05160=1040.627,57.852,413.366,169.673,38.079,157.163
C05161=1040.620,57.602,413.384,169.670,38.078,157.163
C05162=1040.615,57.353,413.401,169.668,38.077,157.163
C05163=1040.608,57.104,413.419,169.666,38.077,157.163
C05164=1040.601,56.854,413.436,169.664,38.076,157.163
C05165=1040.595,56.605,413.453,169.663,38.075,157.163
C05166=1040.589,56.356,413.471,169.661,38.074,157.162
C05167=1040.583,56.107,413.488,169.659,38.074,157.162
C05168=1040.576,55.857,413.506,169.656,38.073,157.162
C05169=1040.569,55.608,413.523,169.654,38.073,157.162
C05170=1040.564,55.359,413.541,169.653,38.071,157.162
C05171=1040.557,55.109,413.558,169.651,38.071,157.161
C05172=1040.551,54.860,413.574,169.649,38.070,157.161
C05173=1040.545,54.610,413.592,169.647,38.070,157.161
C05174=1040.538,54.361,413.609,169.645,38.069,157.161
C05175=1040.533,54.112,413.627,169.642,38.068,157.161
C05176=1040.526,53.862,413.644,169.641,38.067,157.161
C05177=1040.519,53.614,413.661,169.639,38.067,157.161
C05178=1040.513,53.364,413.679,169.637,38.066,157.160
C05179=1040.506,53.114,413.697,169.635,38.065,157.160
C05180=1040.500,52.866,413.714,169.633,38.064,157.160
C05181=1040.494,52.615,413.731,169.631,38.064,157.160
C05182=1040.488,52.367,413.748,169.630,38.063,157.160
C05183=1040.481,52.117,413.765,169.627,38.063,157.160
C05184=1040.476,51.868,413.783,169.625,38.062,157.159
C05185=1040.469,51.619,413.800,169.623,38.061,157.159
C05186=1040.463,51.370,413.817,169.621,38.060,157.159
C05187=1040.457,51.120,413.834,169.620,38.060,157.159
C05188=1040.451,50.871,413.851,169.618,38.059,157.159
C05189=1040.444,50.621,413.868,169.616,38.058,157.158
C05190=1040.438,50.372,413.886,169.614,38.057,157.158
C05191=1040.431,50.123,413.903,169.611,38.057,157.158
C05192=1040.425,49.873,413.920,169.609,38.056,157.158
C05193=1040.419,49.624,413.938,169.608,38.055,157.158
C05194=1040.412,49.374,413.955,169.606,38.055,157.158
C05195=1040.406,49.126,413.972,169.604,38.053,157.157
C05196=1040.400,48.875,413.989,169.602,38.053,157.157
C05197=1040.394,48.627,414.006,169.600,38.052,157.157
C05198=1040.387,48.377,414.023,169.598,38.052,157.157
C05199=1040.382,48.128,414.041,169.596,38.050,157.157
C05200=1040.376,47.879,414.057,169.594,38.050,157.157
C05201=1040.369,47.629,414.075,169.592,38.049,157.156
C05202=1040.363,47.380,414.092,169.590,38.049,157.156
C05203=1040.357,47.130,414.109,169.589,38.048,157.156
C05204=1040.351,46.882,414.126,169.587,38.047,157.156
C05205=1040.344,46.632,414.144,169.584,38.046,157.156
C05206=1040.338,46.383,414.161,169.582,38.045,157.156
C05207=1040.332,46.133,414.177,169.580,38.045,157.155
C05208=1040.326,45.884,414.195,169.578,38.044,157.155
C05209=1040.320,45.635,414.211,169.577,38.044,157.155
C05210=1040.313,45.385,414.228,169.575,38.042,157.155
C05211=1040.306,45.099,414.248,169.573,38.042,157.155
C05212=1040.299,44.812,414.268,169.570,38.041,157.154
C05213=1040.292,44.526,414.287,169.568,38.040,157.154
C05214=1040.285,44.240,414.307,169.565,38.039,157.154
C05215=1040.279,43.990,414.324,169.564,38.038,157.154
C05216=1040.273,43.741,414.341,169.562,38.038,157.154
C05217=1040.267,43.490,414.358,169.560,38.037,157.154
C05218=1040.261,43.242,414.375,169.558,38.036,157.153
C05219=1040.254,42.992,414.392,169.555,38.035,157.153
C05220=1040.248,42.743,414.409,169.553,38.035,157.153
C05221=1040.242,42.494,414.425,169.552,38.034,157.153
C05222=1040.235,42.244,414.442,169.550,38.034,157.153
C05223=1040.229,41.995,414.458,169.548,38.033,157.153
C05224=1040.222,41.745,414.476,169.546,38.032,157.152
C05225=1040.216,41.496,414.492,169.544,38.031,157.152
C05226=1040.210,41.247,414.509,169.542,38.031,157.152
C05227=1040.203,40.997,414.526,169.540,38.030,157.152
C05228=1040.198,40.748,414.543,169.538,38.030,157.152
C05229=1040.191,40.498,414.560,169.536,38.028,157.152
C05230=1040.185,40.249,414.577,169.534,38.028,157.151
C05231=1040.179,40.000,414.593,169.532,38.027,157.151
C05232=1040.172,39.751,414.610,169.530,38.027,157.151
C05233=1040.166,39.501,414.627,169.528,38.026,157.151
C05234=1040.160,39.251,414.643,169.527,38.026,157.151
C05235=1040.153,39.003,414.660,169.524,38.024,157.151
C05236=1040.148,38.753,414.676,169.522,38.024,157.151
C05237=1040.141,38.504,414.694,169.520,38.023,157.150
C05238=1040.135,38.254,414.710,169.518,38.023,157.150
C05239=1040.129,38.005,414.726,169.516,38.022,157.150
C05240=1040.122,37.756,414.744,169.514,38.021,157.150
C05241=1040.116,37.506,414.760,169.513,38.020,157.150
C05242=1040.110,37.257,414.776,169.511,38.020,157.150
C05243=1040.103,37.007,414.793,169.508,38.019,157.149
C05244=1040.097,36.758,414.810,169.506,38.019,157.149
C05245=1040.090,36.509,414.825,169.504,38.018,157.149
C05246=1040.084,36.260,414.843,169.502,38.018,157.149
C05247=1040.078,36.010,414.859,169.500,38.017,157.149
C05248=1040.071,35.760,414.876,169.498,38.016,157.149
C05249=1040.065,35.511,414.892,169.497,38.016,157.149
C05250=1040.058,35.263,414.908,169.495,38.015,157.148
C05251=1040.052,35.012,414.925,169.493,38.015,157.148
C05252=1040.046,34.763,414.941,169.490,38.014,157.148
C05253=1040.040,34.514,414.957,169.488,38.013,157.148
C05254=1040.033,34.264,414.974,169.486,38.012,157.148
C05255=1040.026,34.015,414.990,169.484,38.012,157.148
C05256=1040.020,33.766,415.007,169.482,38.011,157.147
C05257=1040.014,33.517,415.023,169.480,38.011,157.147
C05258=1040.008,33.267,415.040,169.479,38.010,157.147
C05259=1040.002,33.017,415.056,169.477,38.010,157.147
C05260=1039.995,32.769,415.072,169.474,38.009,157.147
C05261=1039.988,32.519,415.089,169.472,38.008,157.147
C05262=1039.982,32.269,415.105,169.470,38.008,157.147
C05263=1039.976,32.020,415.121,169.468,38.007,157.147
C05264=1039.970,31.771,415.138,169.466,38.006,157.146
C05265=1039.963,31.521,415.154,169.464,38.006,157.146
C05266=1039.957,31.272,415.171,169.463,38.005,157.146
C05267=1039.951,31.023,415.187,169.461,38.004,157.146
C05268=1039.944,30.773,415.203,169.459,38.004,157.146
C05269=1039.938,30.523,415.220,169.456,38.003,157.146
C05270=1039.932,30.274,415.235,169.454,38.003,157.145
C05271=1039.926,30.025,415.252,169.452,38.002,157.145
C05272=1039.920,29.776,415.268,169.450,38.002,157.145
C05273=1039.913,29.526,415.284,169.448,38.001,157.145
C05274=1039.907,29.277,415.300,169.446,38.000,157.145
C05275=1039.900,28.990,415.319,169.444,37.999,157.145
C05276=1039.892,28.704,415.338,169.442,37.999,157.144
C05277=1039.885,28.416,415.356,169.439,37.998,157.144
C05278=1039.878,28.130,415.376,169.437,37.997,157.144
C05279=1039.871,27.881,415.391,169.435,37.996,157.144
C05280=1039.866,27.631,415.407,169.433,37.996,157.144
C05281=1039.859,27.382,415.423,169.431,37.995,157.144
C05282=1039.852,27.132,415.440,169.429,37.995,157.144
C05283=1039.846,26.883,415.456,169.427,37.994,157.143
C05284=1039.840,26.634,415.472,169.425,37.994,157.143
C05285=1039.834,26.385,415.488,169.422,37.993,157.143
C05286=1039.826,26.135,415.504,169.420,37.992,157.143
C05287=1039.820,25.885,415.520,169.419,37.992,157.143
C05288=1039.814,25.636,415.536,169.417,37.991,157.143
C05289=1039.808,25.387,415.552,169.415,37.991,157.143
C05290=1039.802,25.137,415.568,169.413,37.990,157.142
C05291=1039.795,24.887,415.584,169.411,37.990,157.142
C05292=1039.789,24.638,415.600,169.409,37.989,157.142
C05293=1039.782,24.389,415.616,169.407,37.988,157.142
C05294=1039.776,24.140,415.632,169.404,37.988,157.142
C05295=1039.770,23.891,415.648,169.402,37.987,157.142
C05296=1039.764,23.641,415.664,169.400,37.987,157.142
C05297=1039.756,23.391,415.680,169.398,37.986,157.141
C05298=1039.751,23.141,415.695,169.396,37.986,157.141
C05299=1039.745,22.892,415.712,169.394,37.985,157.141
C05300=1039.738,22.643,415.727,169.393,37.984,157.141
C05301=1039.732,22.394,415.744,169.391,37.984,157.141
C05302=1039.725,22.145,415.759,169.389,37.983,157.141
C05303=1039.720,21.895,415.775,169.387,37.983,157.141
C05304=1039.712,21.645,415.791,169.384,37.982,157.140
C05305=1039.707,21.396,415.807,169.382,37.982,157.140
C05306=1039.700,21.147,415.823,169.380,37.981,157.140
C05307=1039.694,20.897,415.839,169.378,37.981,157.140
C05308=1039.688,20.648,415.854,169.376,37.980,157.140
C05309=1039.682,20.398,415.870,169.374,37.979,157.140
C05310=1039.675,20.149,415.886,169.372,37.979,157.140
C05311=1039.669,19.900,415.902,169.370,37.978,157.140
C05312=1039.663,19.650,415.917,169.368,37.978,157.139
C05313=1039.656,19.400,415.934,169.365,37.977,157.139
C05314=1039.649,19.151,415.949,169.363,37.977,157.139
C05315=1039.644,18.901,415.965,169.362,37.976,157.139
C05316=1039.637,18.652,415.981,169.360,37.975,157.139
C05317=1039.630,18.403,415.996,169.358,37.975,157.139
C05318=1039.624,18.154,416.012,169.356,37.974,157.139
C05319=1039.618,17.904,416.027,169.354,37.974,157.138
C05320=1039.611,17.655,416.043,169.352,37.973,157.138
C05321=1039.606,17.405,416.059,169.350,37.973,157.138
C05322=1039.599,17.156,416.074,169.347,37.972,157.138
C05323=1039.593,16.907,416.090,169.345,37.971,157.138
C05324=1039.586,16.656,416.106,169.343,37.971,157.138
C05325=1039.579,16.407,416.121,169.341,37.970,157.138
C05326=1039.573,16.158,416.138,169.339,37.970,157.137
C05327=1039.567,15.908,416.153,169.337,37.969,157.137
C05328=1039.560,15.659,416.168,169.335,37.969,157.137
C05329=1039.555,15.409,416.184,169.333,37.968,157.137
C05330=1039.548,15.160,416.200,169.331,37.968,157.137
C05331=1039.542,14.911,416.216,169.329,37.968,157.137
C05332=1039.536,14.661,416.231,169.326,37.967,157.137
C05333=1039.529,14.412,416.246,169.324,37.966,157.137
C05334=1039.523,14.162,416.262,169.322,37.966,157.136
C05335=1039.517,13.913,416.278,169.320,37.965,157.136
C05336=1039.510,13.664,416.293,169.318,37.965,157.136
C05337=1039.503,13.415,416.308,169.316,37.964,157.136
C05338=1039.497,13.165,416.323,169.314,37.964,157.136
C05339=1039.490,12.880,416.341,169.312,37.963,157.136
C05340=1039.483,12.594,416.359,169.310,37.962,157.136
C05341=1039.476,12.308,416.376,169.307,37.962,157.135
C05342=1039.468,12.023,416.394,169.304,37.961,157.135
C05343=1039.461,11.774,416.409,169.302,37.961,157.135
C05344=1039.455,11.524,416.424,169.300,37.961,157.135
C05345=1039.449,11.275,416.439,169.298,37.960,157.135
C05346=1039.442,11.026,416.455,169.296,37.960,157.135
C05347=1039.435,10.776,416.470,169.294,37.959,157.135
C05348=1039.429,10.527,416.486,169.292,37.959,157.135
C05349=1039.422,10.277,416.501,169.290,37.959,157.135
C05350=1039.417,10.027,416.516,169.288,37.958,157.134
C05351=1039.410,9.778,416.532,169.286,37.958,157.134
C05352=1039.404,9.529,416.547,169.284,37.957,157.134
C05353=1039.397,9.279,416.562,169.281,37.956,157.134
C05354=1039.391,9.030,416.577,169.279,37.956,157.134
C05355=1039.384,8.780,416.592,169.277,37.956,157.134
C05356=1039.378,8.531,416.607,169.275,37.955,157.134
C05357=1039.371,8.282,416.623,169.273,37.955,157.134
C05358=1039.365,8.032,416.638,169.271,37.954,157.133
C05359=1039.358,7.782,416.653,169.269,37.954,157.133
C05360=1039.352,7.533,416.669,169.267,37.953,157.133
C05361=1039.346,7.283,416.684,169.265,37.953,157.133
C05362=1039.340,7.034,416.699,169.263,37.953,157.133
C05363=1039.334,6.785,416.713,169.261,37.952,157.133
C05364=1039.327,6.536,416.729,169.258,37.951,157.133
C05365=1039.321,6.286,416.744,169.256,37.951,157.133
C05366=1039.314,6.036,416.759,169.254,37.950,157.133
C05367=1039.308,5.787,416.774,169.252,37.950,157.132
C05368=1039.301,5.538,416.790,169.250,37.949,157.132
C05369=1039.295,5.288,416.805,169.248,37.949,157.132
C05370=1039.289,5.038,416.820,169.246,37.949,157.132
C05371=1039.282,4.789,416.834,169.244,37.948,157.132
C05372=1039.276,4.540,416.850,169.242,37.948,157.132
C05373=1039.270,4.290,416.865,169.240,37.947,157.132
C05374=1039.264,4.041,416.880,169.237,37.946,157.132
C05375=1039.258,3.791,416.895,169.235,37.946,157.131
C05376=1039.251,3.541,416.910,169.233,37.946,157.131
C05377=1039.245,3.292,416.925,169.231,37.945,157.131
C05378=1039.238,3.043,416.941,169.229,37.945,157.131
C05379=1039.232,2.794,416.955,169.227,37.944,157.131
C05380=1039.226,2.544,416.970,169.225,37.944,157.131
C05381=1039.220,2.294,416.985,169.223,37.943,157.131
C05382=1039.213,2.045,417.000,169.221,37.943,157.131
C05383=1039.207,1.795,417.015,169.219,37.943,157.131
C05384=1039.201,1.545,417.030,169.217,37.942,157.130
C05385=1039.195,1.296,417.045,169.214,37.941,157.130
C05386=1039.188,1.047,417.060,169.212,37.941,157.130
C05387=1039.182,0.798,417.075,169.210,37.940,157.130
C05388=1039.175,0.548,417.090,169.208,37.940,157.130
C05389=1039.169,0.298,417.105,169.206,37.939,157.130
C05390=1039.163,0.050,417.120,169.204,37.939,157.130
C05391=1039.157,-0.200,417.135,169.201,37.939,157.130
C05392=1039.150,-0.450,417.150,169.199,37.938,157.129
C05393=1039.144,-0.699,417.165,169.197,37.938,157.129
C05394=1039.139,-0.949,417.180,169.195,37.937,157.129
C05395=1039.133,-1.198,417.195,169.192,37.936,157.129
C05396=1039.126,-1.448,417.210,169.190,37.936,157.129
C05397=1039.120,-1.698,417.225,169.188,37.935,157.129
C05398=1039.113,-1.947,417.240,169.186,37.935,157.129
C05399=1039.108,-2.196,417.254,169.184,37.934,157.128
C05400=1039.101,-2.446,417.269,169.182,37.934,157.128
C05401=1039.095,-2.696,417.284,169.180,37.934,157.128
C05402=1039.089,-2.945,417.299,169.178,37.933,157.128
C05403=1039.081,-3.229,417.315,169.176,37.933,157.128
C05404=1039.074,-3.512,417.332,169.173,37.932,157.128
C05405=1039.067,-3.795,417.349,169.170,37.931,157.128
C05406=1039.060,-4.079,417.365,169.168,37.931,157.128
C05407=1039.054,-4.328,417.380,169.166,37.931,157.128
C05408=1039.047,-4.578,417.395,169.164,37.930,157.127
C05409=1039.041,-4.827,417.410,169.161,37.930,157.127
C05410=1039.034,-5.076,417.424,169.159,37.929,157.127
C05411=1039.028,-5.326,417.438,169.157,37.929,157.127
C05412=1039.022,-5.576,417.453,169.155,37.929,157.127
C05413=1039.015,-5.825,417.467,169.153,37.928,157.127
C05414=1039.009,-6.074,417.482,169.151,37.928,157.127
C05415=1039.002,-6.324,417.497,169.149,37.928,157.127
C05416=1038.995,-6.573,417.511,169.147,37.927,157.127
C05417=1038.990,-6.823,417.525,169.145,37.927,157.127
C05418=1038.983,-7.073,417.540,169.142,37.927,157.126
C05419=1038.977,-7.322,417.555,169.139,37.926,157.126
C05420=1038.970,-7.572,417.569,169.137,37.926,157.126
C05421=1038.965,-7.821,417.583,169.135,37.926,157.126
C05422=1038.958,-8.071,417.598,169.133,37.925,157.126
C05423=1038.951,-8.320,417.613,169.131,37.925,157.126
C05424=1038.945,-8.569,417.627,169.129,37.925,157.126
C05425=1038.939,-8.819,417.641,169.127,37.924,157.126
C05426=1038.932,-9.069,417.656,169.125,37.923,157.126
C05427=1038.926,-9.318,417.670,169.123,37.923,157.126
C05428=1038.920,-9.568,417.685,169.121,37.923,157.125
C05429=1038.913,-9.817,417.699,169.118,37.922,157.125
C05430=1038.907,-10.066,417.713,169.116,37.922,157.125
C05431=1038.901,-10.317,417.728,169.113,37.922,157.125
C05432=1038.894,-10.566,417.742,169.111,37.921,157.125
C05433=1038.888,-10.815,417.757,169.109,37.921,157.125
C05434=1038.882,-11.065,417.771,169.107,37.921,157.125
C05435=1038.876,-11.314,417.785,169.105,37.920,157.125
C05436=1038.869,-11.563,417.800,169.103,37.920,157.125
C05437=1038.863,-11.814,417.814,169.101,37.920,157.124
C05438=1038.857,-12.062,417.828,169.098,37.919,157.124
C05439=1038.850,-12.312,417.843,169.096,37.919,157.124
C05440=1038.844,-12.562,417.857,169.094,37.919,157.124
C05441=1038.838,-12.811,417.871,169.092,37.918,157.124
C05442=1038.832,-13.061,417.885,169.090,37.918,157.124
C05443=1038.826,-13.310,417.900,169.088,37.918,157.124
C05444=1038.819,-13.560,417.914,169.085,37.917,157.124
C05445=1038.813,-13.809,417.928,169.083,37.916,157.124
C05446=1038.807,-14.059,417.943,169.080,37.916,157.123
C05447=1038.800,-14.309,417.957,169.078,37.916,157.123
C05448=1038.794,-14.558,417.971,169.076,37.915,157.123
C05449=1038.787,-14.808,417.985,169.074,37.915,157.123
C05450=1038.782,-15.057,418.000,169.072,37.915,157.123
C05451=1038.776,-15.307,418.014,169.070,37.914,157.123
C05452=1038.769,-15.556,418.028,169.068,37.914,157.123
C05453=1038.763,-15.806,418.042,169.065,37.914,157.123
C05454=1038.756,-16.055,418.056,169.063,37.913,157.123
C05455=1038.750,-16.304,418.070,169.061,37.913,157.123
C05456=1038.743,-16.554,418.085,169.059,37.913,157.123
C05457=1038.737,-16.803,418.098,169.057,37.913,157.123
C05458=1038.731,-17.054,418.112,169.054,37.912,157.122
C05459=1038.724,-17.302,418.126,169.051,37.912,157.122
C05460=1038.718,-17.552,418.140,169.049,37.912,157.122
C05461=1038.711,-17.802,418.155,169.047,37.911,157.122
C05462=1038.705,-18.051,418.168,169.045,37.911,157.122
C05463=1038.699,-18.301,418.182,169.043,37.911,157.122
C05464=1038.692,-18.550,418.196,169.041,37.911,157.122
C05465=1038.686,-18.800,418.210,169.038,37.910,157.122
C05466=1038.680,-19.050,418.224,169.036,37.910,157.122
